ABB RAPID module: P106.mod

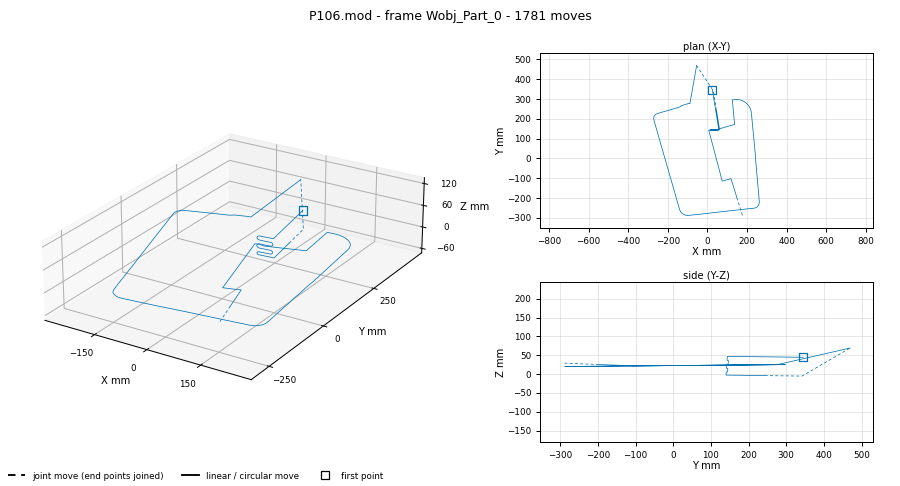
[picture p0: tool path of P106.mod in frame Wobj_Part_0, 1781 of 1791 moves have a stored position in this frame; points joined in program order, loops and branches not executed]
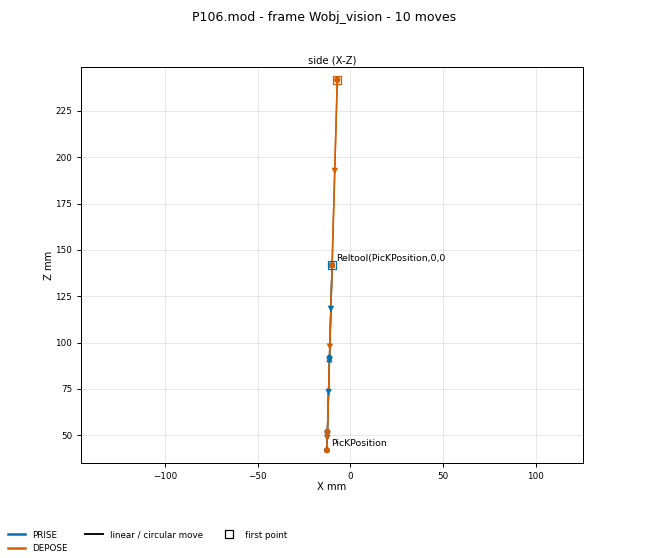
[picture p1: tool path of P106.mod in frame Wobj_vision, 10 of 1791 moves have a stored position in this frame; points joined in program order, loops and branches not executed]
MODULE P106

    ! Nom         :P106
    ! Description :
    ! Créé le     :06/06/2023 16:16:34

    LOCAL CONST SPEEDDATA VitesseLente :=[10,500,0,0];
	LOCAL CONST SPEEDDATA VitesseRapide :=[30,500,0,0];
	LOCAL CONST SPEEDDATA VitesseTronconnage :=[2,500,0,0];
	LOCAL CONST SPEEDDATA VitesseTronconnageApp :=[10,500,0,0];
    !
    !Point de prise
    LOCAL PERS Robtarget PicKPosition := [[-12.6362620334208,-14.9745689455813,41.8593448105357],[-0.00913162142581617,0.993890068091212,0.109216713362201,-0.0130711729443154],[0,0,0,0],[8.999999E+09,8.999999E+09,8.999999E+09,8.999999E+09,8.999999E+09,8.999999E+09]];
	LOCAL PERS Pose Ref := [[0,0,0],[1,0,0,0]];
    !
    !Declaration des points de meulage

    !Tr_meulage_motif_1 : Meulage d'un motif
    LOCAL CONST Robtarget Tr_meulage_motif_1_0 := [[57.250015625,147.518171875,47.0711640625],[0.0569478960959874,-0.0562129652335629,0.700246962774789,-0.709402023393347],[0,0,0,0],[8.999999E+09,8.999999E+09,8.999999E+09,8.999999E+09,8.999999E+09,8.999999E+09]];
    LOCAL CONST Robtarget Tr_meulage_motif_1_1 := [[56.253921875,147.429890625,47.0709765625],[0.0569478960959874,-0.0562129652335629,0.700246962774789,-0.709402023393347],[0,0,0,0],[8.999999E+09,8.999999E+09,8.999999E+09,8.999999E+09,8.999999E+09,8.999999E+09]];
    LOCAL CONST Robtarget Tr_meulage_motif_1_2 := [[55.257828125,147.34159375,47.0707890625],[0.0569478960959874,-0.0562129652335629,0.700246962774789,-0.709402023393347],[0,0,0,0],[8.999999E+09,8.999999E+09,8.999999E+09,8.999999E+09,8.999999E+09,8.999999E+09]];
    LOCAL CONST Robtarget Tr_meulage_motif_1_3 := [[54.261734375,147.253296875,47.07059765625],[0.0569478960959874,-0.0562129652335629,0.700246962774789,-0.709402023393347],[0,0,0,0],[8.999999E+09,8.999999E+09,8.999999E+09,8.999999E+09,8.999999E+09,8.999999E+09]];
    LOCAL CONST Robtarget Tr_meulage_motif_1_4 := [[53.265640625,147.165,47.07041015625],[0.0569478960959874,-0.0562129652335629,0.700246962774789,-0.709402023393347],[0,0,0,0],[8.999999E+09,8.999999E+09,8.999999E+09,8.999999E+09,8.999999E+09,8.999999E+09]];
    LOCAL CONST Robtarget Tr_meulage_motif_1_5 := [[52.269546875,147.076703125,47.07021875],[0.0569478960959874,-0.0562129652335629,0.700246962774789,-0.709402023393347],[0,0,0,0],[8.999999E+09,8.999999E+09,8.999999E+09,8.999999E+09,8.999999E+09,8.999999E+09]];
    LOCAL CONST Robtarget Tr_meulage_motif_1_6 := [[51.27344921875,146.98840625,47.07003125],[0.0569478960959874,-0.0562129652335629,0.700246962774789,-0.709402023393347],[0,0,0,0],[8.999999E+09,8.999999E+09,8.999999E+09,8.999999E+09,8.999999E+09,8.999999E+09]];
    LOCAL CONST Robtarget Tr_meulage_motif_1_7 := [[50.27735546875,146.900125,47.06984375],[0.0569478960959874,-0.0562129652335629,0.700246962774789,-0.709402023393347],[0,0,0,0],[8.999999E+09,8.999999E+09,8.999999E+09,8.999999E+09,8.999999E+09,8.999999E+09]];
    LOCAL CONST Robtarget Tr_meulage_motif_1_8 := [[49.28126171875,146.811828125,47.06965234375],[0.0569478960959874,-0.0562129652335629,0.700246962774789,-0.709402023393347],[0,0,0,0],[8.999999E+09,8.999999E+09,8.999999E+09,8.999999E+09,8.999999E+09,8.999999E+09]];
    LOCAL CONST Robtarget Tr_meulage_motif_1_9 := [[48.28516796875,146.72353125,47.06946484375],[0.0569478960959874,-0.0562129652335629,0.700246962774789,-0.709402023393347],[0,0,0,0],[8.999999E+09,8.999999E+09,8.999999E+09,8.999999E+09,8.999999E+09,8.999999E+09]];
    LOCAL CONST Robtarget Tr_meulage_motif_1_10 := [[47.28907421875,146.635234375,47.0692734375],[0.0569478960959874,-0.0562129652335629,0.700246962774789,-0.709402023393347],[0,0,0,0],[8.999999E+09,8.999999E+09,8.999999E+09,8.999999E+09,8.999999E+09,8.999999E+09]];
    LOCAL CONST Robtarget Tr_meulage_motif_1_11 := [[46.29298046875,146.5469375,47.0690859375],[0.0569478960959874,-0.0562129652335629,0.700246962774789,-0.709402023393347],[0,0,0,0],[8.999999E+09,8.999999E+09,8.999999E+09,8.999999E+09,8.999999E+09,8.999999E+09]];
    LOCAL CONST Robtarget Tr_meulage_motif_1_12 := [[45.2968828125,146.458640625,47.0688984375],[0.0569478960959874,-0.0562129652335629,0.700246962774789,-0.709402023393347],[0,0,0,0],[8.999999E+09,8.999999E+09,8.999999E+09,8.999999E+09,8.999999E+09,8.999999E+09]];
    LOCAL CONST Robtarget Tr_meulage_motif_1_13 := [[44.3007890625,146.370359375,47.06870703125],[0.0569478960959874,-0.0562129652335629,0.700246962774789,-0.709402023393347],[0,0,0,0],[8.999999E+09,8.999999E+09,8.999999E+09,8.999999E+09,8.999999E+09,8.999999E+09]];
    LOCAL CONST Robtarget Tr_meulage_motif_1_14 := [[43.3046953125,146.2820625,47.06851953125],[0.0569478960959874,-0.0562129652335629,0.700246962774789,-0.709402023393347],[0,0,0,0],[8.999999E+09,8.999999E+09,8.999999E+09,8.999999E+09,8.999999E+09,8.999999E+09]];
    LOCAL CONST Robtarget Tr_meulage_motif_1_15 := [[42.3086015625,146.193765625,47.06833203125],[0.0569478960959874,-0.0562129652335629,0.700246962774789,-0.709402023393347],[0,0,0,0],[8.999999E+09,8.999999E+09,8.999999E+09,8.999999E+09,8.999999E+09,8.999999E+09]];
    LOCAL CONST Robtarget Tr_meulage_motif_1_16 := [[41.3125078125,146.10546875,47.068140625],[0.0569478960959874,-0.0562129652335629,0.700246962774789,-0.709402023393347],[0,0,0,0],[8.999999E+09,8.999999E+09,8.999999E+09,8.999999E+09,8.999999E+09,8.999999E+09]];
    LOCAL CONST Robtarget Tr_meulage_motif_1_17 := [[40.31641015625,146.017171875,47.067953125],[0.0569478960959874,-0.0562129652335629,0.700246962774789,-0.709402023393347],[0,0,0,0],[8.999999E+09,8.999999E+09,8.999999E+09,8.999999E+09,8.999999E+09,8.999999E+09]];
    LOCAL CONST Robtarget Tr_meulage_motif_1_18 := [[39.32031640625,145.928875,47.06776171875],[0.0569478960959874,-0.0562129652335629,0.700246962774789,-0.709402023393347],[0,0,0,0],[8.999999E+09,8.999999E+09,8.999999E+09,8.999999E+09,8.999999E+09,8.999999E+09]];
    LOCAL CONST Robtarget Tr_meulage_motif_1_19 := [[38.32422265625,145.84059375,47.06757421875],[0.0569478960959874,-0.0562129652335629,0.700246962774789,-0.709402023393347],[0,0,0,0],[8.999999E+09,8.999999E+09,8.999999E+09,8.999999E+09,8.999999E+09,8.999999E+09]];
    LOCAL CONST Robtarget Tr_meulage_motif_1_20 := [[37.32812890625,145.752296875,47.06738671875],[0.0569478960959874,-0.0562129652335629,0.700246962774789,-0.709402023393347],[0,0,0,0],[8.999999E+09,8.999999E+09,8.999999E+09,8.999999E+09,8.999999E+09,8.999999E+09]];
    LOCAL CONST Robtarget Tr_meulage_motif_1_21 := [[36.33203515625,145.664,47.0671953125],[0.0569478960959874,-0.0562129652335629,0.700246962774789,-0.709402023393347],[0,0,0,0],[8.999999E+09,8.999999E+09,8.999999E+09,8.999999E+09,8.999999E+09,8.999999E+09]];
    LOCAL CONST Robtarget Tr_meulage_motif_1_22 := [[35.33594140625,145.575703125,47.0670078125],[0.0569478960959874,-0.0562129652335629,0.700246962774789,-0.709402023393347],[0,0,0,0],[8.999999E+09,8.999999E+09,8.999999E+09,8.999999E+09,8.999999E+09,8.999999E+09]];
    LOCAL CONST Robtarget Tr_meulage_motif_1_23 := [[34.33984375,145.48740625,47.06681640625],[0.0569478960959874,-0.0562129652335629,0.700246962774789,-0.709402023393347],[0,0,0,0],[8.999999E+09,8.999999E+09,8.999999E+09,8.999999E+09,8.999999E+09,8.999999E+09]];
    LOCAL CONST Robtarget Tr_meulage_motif_1_24 := [[33.34375,145.399125,47.06662890625],[0.0569478960959874,-0.0562129652335629,0.700246962774789,-0.709402023393347],[0,0,0,0],[8.999999E+09,8.999999E+09,8.999999E+09,8.999999E+09,8.999999E+09,8.999999E+09]];
    LOCAL CONST Robtarget Tr_meulage_motif_1_25 := [[32.34765625,145.310828125,47.06644140625],[0.0569478960959874,-0.0562129652335629,0.700246962774789,-0.709402023393347],[0,0,0,0],[8.999999E+09,8.999999E+09,8.999999E+09,8.999999E+09,8.999999E+09,8.999999E+09]];
    LOCAL CONST Robtarget Tr_meulage_motif_1_26 := [[31.3515625,145.22253125,47.06625],[0.0569478960959874,-0.0562129652335629,0.700246962774789,-0.709402023393347],[0,0,0,0],[8.999999E+09,8.999999E+09,8.999999E+09,8.999999E+09,8.999999E+09,8.999999E+09]];
    LOCAL CONST Robtarget Tr_meulage_motif_1_27 := [[30.35546875,145.134234375,47.0660625],[0.0569478960959874,-0.0562129652335629,0.700246962774789,-0.709402023393347],[0,0,0,0],[8.999999E+09,8.999999E+09,8.999999E+09,8.999999E+09,8.999999E+09,8.999999E+09]];
    LOCAL CONST Robtarget Tr_meulage_motif_1_28 := [[29.359373046875,145.0459375,47.06587109375],[0.0569478960959874,-0.0562129652335629,0.700246962774789,-0.709402023393347],[0,0,0,0],[8.999999E+09,8.999999E+09,8.999999E+09,8.999999E+09,8.999999E+09,8.999999E+09]];
    LOCAL CONST Robtarget Tr_meulage_motif_1_29 := [[28.363279296875,144.957640625,47.06568359375],[0.0569478960959874,-0.0562129652335629,0.700246962774789,-0.709402023393347],[0,0,0,0],[8.999999E+09,8.999999E+09,8.999999E+09,8.999999E+09,8.999999E+09,8.999999E+09]];
    LOCAL CONST Robtarget Tr_meulage_motif_1_30 := [[27.36718359375,144.869359375,47.06549609375],[0.0569478960959874,-0.0562129652335629,0.700246962774789,-0.709402023393347],[0,0,0,0],[8.999999E+09,8.999999E+09,8.999999E+09,8.999999E+09,8.999999E+09,8.999999E+09]];
    LOCAL CONST Robtarget Tr_meulage_motif_1_31 := [[26.37108984375,144.7810625,47.0653046875],[0.0569478960959874,-0.0562129652335629,0.700246962774789,-0.709402023393347],[0,0,0,0],[8.999999E+09,8.999999E+09,8.999999E+09,8.999999E+09,8.999999E+09,8.999999E+09]];
    LOCAL CONST Robtarget Tr_meulage_motif_1_32 := [[25.37499609375,144.692765625,47.0651171875],[0.0569478960959874,-0.0562129652335629,0.700246962774789,-0.709402023393347],[0,0,0,0],[8.999999E+09,8.999999E+09,8.999999E+09,8.999999E+09,8.999999E+09,8.999999E+09]];
    LOCAL CONST Robtarget Tr_meulage_motif_1_33 := [[24.378900390625,144.60446875,47.06492578125],[0.0569478960959874,-0.0562129652335629,0.700246962774789,-0.709402023393347],[0,0,0,0],[8.999999E+09,8.999999E+09,8.999999E+09,8.999999E+09,8.999999E+09,8.999999E+09]];
    LOCAL CONST Robtarget Tr_meulage_motif_1_34 := [[23.382806640625,144.516171875,47.06473828125],[0.0569478960959874,-0.0562129652335629,0.700246962774789,-0.709402023393347],[0,0,0,0],[8.999999E+09,8.999999E+09,8.999999E+09,8.999999E+09,8.999999E+09,8.999999E+09]];
    LOCAL CONST Robtarget Tr_meulage_motif_1_35 := [[22.386712890625,144.427875,47.06455078125],[0.0569478960959874,-0.0562129652335629,0.700246962774789,-0.709402023393347],[0,0,0,0],[8.999999E+09,8.999999E+09,8.999999E+09,8.999999E+09,8.999999E+09,8.999999E+09]];
    LOCAL CONST Robtarget Tr_meulage_motif_1_36 := [[21.3906171875,144.33959375,47.064359375],[0.0569478960959874,-0.0562129652335629,0.700246962774789,-0.709402023393347],[0,0,0,0],[8.999999E+09,8.999999E+09,8.999999E+09,8.999999E+09,8.999999E+09,8.999999E+09]];
    LOCAL CONST Robtarget Tr_meulage_motif_1_37 := [[20.3945234375,144.251296875,47.064171875],[0.0569478960959874,-0.0562129652335629,0.700246962774789,-0.709402023393347],[0,0,0,0],[8.999999E+09,8.999999E+09,8.999999E+09,8.999999E+09,8.999999E+09,8.999999E+09]];
    LOCAL CONST Robtarget Tr_meulage_motif_1_38 := [[19.3984296875,144.163,47.06398046875],[0.0569478960959874,-0.0562129652335629,0.700246962774789,-0.709402023393347],[0,0,0,0],[8.999999E+09,8.999999E+09,8.999999E+09,8.999999E+09,8.999999E+09,8.999999E+09]];
    LOCAL CONST Robtarget Tr_meulage_motif_1_39 := [[18.41045703125,144.067546875,46.95348046875],[0.0569478960959874,-0.0562129652335629,0.700246962774789,-0.709402023393347],[0,0,0,0],[8.999999E+09,8.999999E+09,8.999999E+09,8.999999E+09,8.999999E+09,8.999999E+09]];
    LOCAL CONST Robtarget Tr_meulage_motif_1_40 := [[17.469013671875,143.969078125,46.74264453125],[0.0569478960959874,-0.0562129652335629,0.700246962774789,-0.709402023393347],[0,0,0,0],[8.999999E+09,8.999999E+09,8.999999E+09,8.999999E+09,8.999999E+09,8.999999E+09]];
    LOCAL CONST Robtarget Tr_meulage_motif_1_41 := [[16.62137890625,143.87459375,46.47132421875],[0.0569478960959874,-0.0562129652335629,0.700246962774789,-0.709402023393347],[0,0,0,0],[8.999999E+09,8.999999E+09,8.999999E+09,8.999999E+09,8.999999E+09,8.999999E+09]];
    LOCAL CONST Robtarget Tr_meulage_motif_1_42 := [[15.8761484375,143.78890625,46.1959375],[0.0569478960959874,-0.0562129652335629,0.700246962774789,-0.709402023393347],[0,0,0,0],[8.999999E+09,8.999999E+09,8.999999E+09,8.999999E+09,8.999999E+09,8.999999E+09]];
    LOCAL CONST Robtarget Tr_meulage_motif_1_43 := [[14.7833583984375,143.6481875,45.58115234375],[0.0569478960959874,-0.0562129652335629,0.700246962774789,-0.709402023393347],[0,0,0,0],[8.999999E+09,8.999999E+09,8.999999E+09,8.999999E+09,8.999999E+09,8.999999E+09]];
    LOCAL CONST Robtarget Tr_meulage_motif_1_44 := [[13.768947265625,143.497953125,44.7354375],[0.0569478960959874,-0.0562129652335629,0.700246962774789,-0.709402023393347],[0,0,0,0],[8.999999E+09,8.999999E+09,8.999999E+09,8.999999E+09,8.999999E+09,8.999999E+09]];
    LOCAL CONST Robtarget Tr_meulage_motif_1_45 := [[12.9312021484375,143.350828125,43.7139765625],[0.0569478960959874,-0.0562129652335629,0.700246962774789,-0.709402023393347],[0,0,0,0],[8.999999E+09,8.999999E+09,8.999999E+09,8.999999E+09,8.999999E+09,8.999999E+09]];
    LOCAL CONST Robtarget Tr_meulage_motif_1_46 := [[12.4521484375,143.228921875,42.60050390625],[0.0569478960959874,-0.0562129652335629,0.700246962774789,-0.709402023393347],[0,0,0,0],[8.999999E+09,8.999999E+09,8.999999E+09,8.999999E+09,8.999999E+09,8.999999E+09]];
    LOCAL CONST Robtarget Tr_meulage_motif_1_47 := [[12.429677734375,143.17740625,41.90628125],[0.0569478960959874,-0.0562129652335629,0.700246962774789,-0.709402023393347],[0,0,0,0],[8.999999E+09,8.999999E+09,8.999999E+09,8.999999E+09,8.999999E+09,8.999999E+09]];
    LOCAL CONST Robtarget Tr_meulage_motif_1_48 := [[12.43394140625,143.13071875,41.2466953125],[0.0569478960959874,-0.0562129652335629,0.700246962774789,-0.709402023393347],[0,0,0,0],[8.999999E+09,8.999999E+09,8.999999E+09,8.999999E+09,8.999999E+09,8.999999E+09]];
    LOCAL CONST Robtarget Tr_meulage_motif_1_49 := [[12.49286328125,143.08890625,40.58727734375],[0.0569478960959874,-0.0562129652335629,0.700246962774789,-0.709402023393347],[0,0,0,0],[8.999999E+09,8.999999E+09,8.999999E+09,8.999999E+09,8.999999E+09,8.999999E+09]];
    LOCAL CONST Robtarget Tr_meulage_motif_1_50 := [[12.9962392578125,143.055109375,39.488390625],[0.0569478960959874,-0.0562129652335629,0.700246962774789,-0.709402023393347],[0,0,0,0],[8.999999E+09,8.999999E+09,8.999999E+09,8.999999E+09,8.999999E+09,8.999999E+09]];
    LOCAL CONST Robtarget Tr_meulage_motif_1_51 := [[13.8560078125,143.0596875,38.4844609375],[0.0569478960959874,-0.0562129652335629,0.700246962774789,-0.709402023393347],[0,0,0,0],[8.999999E+09,8.999999E+09,8.999999E+09,8.999999E+09,8.999999E+09,8.999999E+09]];
    LOCAL CONST Robtarget Tr_meulage_motif_1_52 := [[14.8807607421875,143.09153125,37.65786328125],[0.0569478960959874,-0.0562129652335629,0.700246962774789,-0.709402023393347],[0,0,0,0],[8.999999E+09,8.999999E+09,8.999999E+09,8.999999E+09,8.999999E+09,8.999999E+09]];
    LOCAL CONST Robtarget Tr_meulage_motif_1_53 := [[15.56772265625,143.124265625,37.26323828125],[0.0569478960959874,-0.0562129652335629,0.700246962774789,-0.709402023393347],[0,0,0,0],[8.999999E+09,8.999999E+09,8.999999E+09,8.999999E+09,8.999999E+09,8.999999E+09]];
    LOCAL CONST Robtarget Tr_meulage_motif_1_54 := [[16.724498046875,143.192109375,36.77715234375],[0.0569478960959874,-0.0562129652335629,0.700246962774789,-0.709402023393347],[0,0,0,0],[8.999999E+09,8.999999E+09,8.999999E+09,8.999999E+09,8.999999E+09,8.999999E+09]];
    LOCAL CONST Robtarget Tr_meulage_motif_1_55 := [[17.567931640625,143.248078125,36.5138828125],[0.0569478960959874,-0.0562129652335629,0.700246962774789,-0.709402023393347],[0,0,0,0],[8.999999E+09,8.999999E+09,8.999999E+09,8.999999E+09,8.999999E+09,8.999999E+09]];
    LOCAL CONST Robtarget Tr_meulage_motif_1_56 := [[18.497609375,143.3159375,36.31010546875],[0.0569478960959874,-0.0562129652335629,0.700246962774789,-0.709402023393347],[0,0,0,0],[8.999999E+09,8.999999E+09,8.999999E+09,8.999999E+09,8.999999E+09,8.999999E+09]];
    LOCAL CONST Robtarget Tr_meulage_motif_1_57 := [[19.4760390625,143.3949375,36.20197265625],[0.0569478960959874,-0.0562129652335629,0.700246962774789,-0.709402023393347],[0,0,0,0],[8.999999E+09,8.999999E+09,8.999999E+09,8.999999E+09,8.999999E+09,8.999999E+09]];
    LOCAL CONST Robtarget Tr_meulage_motif_1_58 := [[20.4654375,143.474765625,36.09184375],[0.0569478960959874,-0.0562129652335629,0.700246962774789,-0.709402023393347],[0,0,0,0],[8.999999E+09,8.999999E+09,8.999999E+09,8.999999E+09,8.999999E+09,8.999999E+09]];
    LOCAL CONST Robtarget Tr_meulage_motif_1_59 := [[21.461533203125,143.5630625,36.09203125],[0.0569478960959874,-0.0562129652335629,0.700246962774789,-0.709402023393347],[0,0,0,0],[8.999999E+09,8.999999E+09,8.999999E+09,8.999999E+09,8.999999E+09,8.999999E+09]];
    LOCAL CONST Robtarget Tr_meulage_motif_1_60 := [[22.457626953125,143.65134375,36.09222265625],[0.0569478960959874,-0.0562129652335629,0.700246962774789,-0.709402023393347],[0,0,0,0],[8.999999E+09,8.999999E+09,8.999999E+09,8.999999E+09,8.999999E+09,8.999999E+09]];
    LOCAL CONST Robtarget Tr_meulage_motif_1_61 := [[23.453720703125,143.739640625,36.09241015625],[0.0569478960959874,-0.0562129652335629,0.700246962774789,-0.709402023393347],[0,0,0,0],[8.999999E+09,8.999999E+09,8.999999E+09,8.999999E+09,8.999999E+09,8.999999E+09]];
    LOCAL CONST Robtarget Tr_meulage_motif_1_62 := [[24.44981640625,143.8279375,36.0926015625],[0.0569478960959874,-0.0562129652335629,0.700246962774789,-0.709402023393347],[0,0,0,0],[8.999999E+09,8.999999E+09,8.999999E+09,8.999999E+09,8.999999E+09,8.999999E+09]];
    LOCAL CONST Robtarget Tr_meulage_motif_1_63 := [[25.44591015625,143.916234375,36.0927890625],[0.0569478960959874,-0.0562129652335629,0.700246962774789,-0.709402023393347],[0,0,0,0],[8.999999E+09,8.999999E+09,8.999999E+09,8.999999E+09,8.999999E+09,8.999999E+09]];
    LOCAL CONST Robtarget Tr_meulage_motif_1_64 := [[26.44200390625,144.00453125,36.0929765625],[0.0569478960959874,-0.0562129652335629,0.700246962774789,-0.709402023393347],[0,0,0,0],[8.999999E+09,8.999999E+09,8.999999E+09,8.999999E+09,8.999999E+09,8.999999E+09]];
    LOCAL CONST Robtarget Tr_meulage_motif_1_65 := [[27.438099609375,144.092828125,36.09316796875],[0.0569478960959874,-0.0562129652335629,0.700246962774789,-0.709402023393347],[0,0,0,0],[8.999999E+09,8.999999E+09,8.999999E+09,8.999999E+09,8.999999E+09,8.999999E+09]];
    LOCAL CONST Robtarget Tr_meulage_motif_1_66 := [[28.434193359375,144.181109375,36.09335546875],[0.0569478960959874,-0.0562129652335629,0.700246962774789,-0.709402023393347],[0,0,0,0],[8.999999E+09,8.999999E+09,8.999999E+09,8.999999E+09,8.999999E+09,8.999999E+09]];
    LOCAL CONST Robtarget Tr_meulage_motif_1_67 := [[29.430287109375,144.26940625,36.093546875],[0.0569478960959874,-0.0562129652335629,0.700246962774789,-0.709402023393347],[0,0,0,0],[8.999999E+09,8.999999E+09,8.999999E+09,8.999999E+09,8.999999E+09,8.999999E+09]];
    LOCAL CONST Robtarget Tr_meulage_motif_1_68 := [[30.4263828125,144.357703125,36.093734375],[0.0569478960959874,-0.0562129652335629,0.700246962774789,-0.709402023393347],[0,0,0,0],[8.999999E+09,8.999999E+09,8.999999E+09,8.999999E+09,8.999999E+09,8.999999E+09]];
    LOCAL CONST Robtarget Tr_meulage_motif_1_69 := [[31.4224765625,144.446,36.093921875],[0.0569478960959874,-0.0562129652335629,0.700246962774789,-0.709402023393347],[0,0,0,0],[8.999999E+09,8.999999E+09,8.999999E+09,8.999999E+09,8.999999E+09,8.999999E+09]];
    LOCAL CONST Robtarget Tr_meulage_motif_1_70 := [[32.4185703125,144.534296875,36.09411328125],[0.0569478960959874,-0.0562129652335629,0.700246962774789,-0.709402023393347],[0,0,0,0],[8.999999E+09,8.999999E+09,8.999999E+09,8.999999E+09,8.999999E+09,8.999999E+09]];
    LOCAL CONST Robtarget Tr_meulage_motif_1_71 := [[33.4146640625,144.622578125,36.09430078125],[0.0569478960959874,-0.0562129652335629,0.700246962774789,-0.709402023393347],[0,0,0,0],[8.999999E+09,8.999999E+09,8.999999E+09,8.999999E+09,8.999999E+09,8.999999E+09]];
    LOCAL CONST Robtarget Tr_meulage_motif_1_72 := [[34.41076171875,144.710875,36.09448828125],[0.0569478960959874,-0.0562129652335629,0.700246962774789,-0.709402023393347],[0,0,0,0],[8.999999E+09,8.999999E+09,8.999999E+09,8.999999E+09,8.999999E+09,8.999999E+09]];
    LOCAL CONST Robtarget Tr_meulage_motif_1_73 := [[35.40685546875,144.799171875,36.0946796875],[0.0569478960959874,-0.0562129652335629,0.700246962774789,-0.709402023393347],[0,0,0,0],[8.999999E+09,8.999999E+09,8.999999E+09,8.999999E+09,8.999999E+09,8.999999E+09]];
    LOCAL CONST Robtarget Tr_meulage_motif_1_74 := [[36.40294921875,144.88746875,36.0948671875],[0.0569478960959874,-0.0562129652335629,0.700246962774789,-0.709402023393347],[0,0,0,0],[8.999999E+09,8.999999E+09,8.999999E+09,8.999999E+09,8.999999E+09,8.999999E+09]];
    LOCAL CONST Robtarget Tr_meulage_motif_1_75 := [[37.39904296875,144.975765625,36.09505859375],[0.0569478960959874,-0.0562129652335629,0.700246962774789,-0.709402023393347],[0,0,0,0],[8.999999E+09,8.999999E+09,8.999999E+09,8.999999E+09,8.999999E+09,8.999999E+09]];
    LOCAL CONST Robtarget Tr_meulage_motif_1_76 := [[38.39513671875,145.0640625,36.09524609375],[0.0569478960959874,-0.0562129652335629,0.700246962774789,-0.709402023393347],[0,0,0,0],[8.999999E+09,8.999999E+09,8.999999E+09,8.999999E+09,8.999999E+09,8.999999E+09]];
    LOCAL CONST Robtarget Tr_meulage_motif_1_77 := [[39.39123046875,145.15234375,36.09543359375],[0.0569478960959874,-0.0562129652335629,0.700246962774789,-0.709402023393347],[0,0,0,0],[8.999999E+09,8.999999E+09,8.999999E+09,8.999999E+09,8.999999E+09,8.999999E+09]];
    LOCAL CONST Robtarget Tr_meulage_motif_1_78 := [[40.387328125,145.240640625,36.095625],[0.0569478960959874,-0.0562129652335629,0.700246962774789,-0.709402023393347],[0,0,0,0],[8.999999E+09,8.999999E+09,8.999999E+09,8.999999E+09,8.999999E+09,8.999999E+09]];
    LOCAL CONST Robtarget Tr_meulage_motif_1_79 := [[41.383421875,145.3289375,36.0958125],[0.0569478960959874,-0.0562129652335629,0.700246962774789,-0.709402023393347],[0,0,0,0],[8.999999E+09,8.999999E+09,8.999999E+09,8.999999E+09,8.999999E+09,8.999999E+09]];
    LOCAL CONST Robtarget Tr_meulage_motif_1_80 := [[42.379515625,145.417234375,36.09600390625],[0.0569478960959874,-0.0562129652335629,0.700246962774789,-0.709402023393347],[0,0,0,0],[8.999999E+09,8.999999E+09,8.999999E+09,8.999999E+09,8.999999E+09,8.999999E+09]];
    LOCAL CONST Robtarget Tr_meulage_motif_1_81 := [[43.375609375,145.50553125,36.09619140625],[0.0569478960959874,-0.0562129652335629,0.700246962774789,-0.709402023393347],[0,0,0,0],[8.999999E+09,8.999999E+09,8.999999E+09,8.999999E+09,8.999999E+09,8.999999E+09]];
    LOCAL CONST Robtarget Tr_meulage_motif_1_82 := [[44.371703125,145.593828125,36.09637890625],[0.0569478960959874,-0.0562129652335629,0.700246962774789,-0.709402023393347],[0,0,0,0],[8.999999E+09,8.999999E+09,8.999999E+09,8.999999E+09,8.999999E+09,8.999999E+09]];
    LOCAL CONST Robtarget Tr_meulage_motif_1_83 := [[45.367796875,145.682109375,36.0965703125],[0.0569478960959874,-0.0562129652335629,0.700246962774789,-0.709402023393347],[0,0,0,0],[8.999999E+09,8.999999E+09,8.999999E+09,8.999999E+09,8.999999E+09,8.999999E+09]];
    LOCAL CONST Robtarget Tr_meulage_motif_1_84 := [[46.36389453125,145.77040625,36.0967578125],[0.0569478960959874,-0.0562129652335629,0.700246962774789,-0.709402023393347],[0,0,0,0],[8.999999E+09,8.999999E+09,8.999999E+09,8.999999E+09,8.999999E+09,8.999999E+09]];
    LOCAL CONST Robtarget Tr_meulage_motif_1_85 := [[47.35998828125,145.858703125,36.09694921875],[0.0569478960959874,-0.0562129652335629,0.700246962774789,-0.709402023393347],[0,0,0,0],[8.999999E+09,8.999999E+09,8.999999E+09,8.999999E+09,8.999999E+09,8.999999E+09]];
    LOCAL CONST Robtarget Tr_meulage_motif_1_86 := [[48.35608203125,145.947,36.09713671875],[0.0569478960959874,-0.0562129652335629,0.700246962774789,-0.709402023393347],[0,0,0,0],[8.999999E+09,8.999999E+09,8.999999E+09,8.999999E+09,8.999999E+09,8.999999E+09]];
    LOCAL CONST Robtarget Tr_meulage_motif_1_87 := [[49.35217578125,146.035296875,36.09732421875],[0.0569478960959874,-0.0562129652335629,0.700246962774789,-0.709402023393347],[0,0,0,0],[8.999999E+09,8.999999E+09,8.999999E+09,8.999999E+09,8.999999E+09,8.999999E+09]];
    LOCAL CONST Robtarget Tr_meulage_motif_1_88 := [[50.34826953125,146.12359375,36.097515625],[0.0569478960959874,-0.0562129652335629,0.700246962774789,-0.709402023393347],[0,0,0,0],[8.999999E+09,8.999999E+09,8.999999E+09,8.999999E+09,8.999999E+09,8.999999E+09]];
    LOCAL CONST Robtarget Tr_meulage_motif_1_89 := [[51.33766796875,146.203421875,35.98738671875],[0.0569478960959874,-0.0562129652335629,0.700246962774789,-0.709402023393347],[0,0,0,0],[8.999999E+09,8.999999E+09,8.999999E+09,8.999999E+09,8.999999E+09,8.999999E+09]];
    LOCAL CONST Robtarget Tr_meulage_motif_1_90 := [[52.2818359375,146.272078125,35.77691015625],[0.0569478960959874,-0.0562129652335629,0.700246962774789,-0.709402023393347],[0,0,0,0],[8.999999E+09,8.999999E+09,8.999999E+09,8.999999E+09,8.999999E+09,8.999999E+09]];
    LOCAL CONST Robtarget Tr_meulage_motif_1_91 := [[53.1329765625,146.328171875,35.50591015625],[0.0569478960959874,-0.0562129652335629,0.700246962774789,-0.709402023393347],[0,0,0,0],[8.999999E+09,8.999999E+09,8.999999E+09,8.999999E+09,8.999999E+09,8.999999E+09]];
    LOCAL CONST Robtarget Tr_meulage_motif_1_92 := [[53.84365625,146.36953125,35.20265625],[0.0569478960959874,-0.0562129652335629,0.700246962774789,-0.709402023393347],[0,0,0,0],[8.999999E+09,8.999999E+09,8.999999E+09,8.999999E+09,8.999999E+09,8.999999E+09]];
    LOCAL CONST Robtarget Tr_meulage_motif_1_93 := [[54.87835546875,146.41409375,34.541984375],[0.0569478960959874,-0.0562129652335629,0.700246962774789,-0.709402023393347],[0,0,0,0],[8.999999E+09,8.999999E+09,8.999999E+09,8.999999E+09,8.999999E+09,8.999999E+09]];
    LOCAL CONST Robtarget Tr_meulage_motif_1_94 := [[55.7825859375,146.4300625,33.64248828125],[0.0569478960959874,-0.0562129652335629,0.700246962774789,-0.709402023393347],[0,0,0,0],[8.999999E+09,8.999999E+09,8.999999E+09,8.999999E+09,8.999999E+09,8.999999E+09]];
    LOCAL CONST Robtarget Tr_meulage_motif_1_95 := [[56.3222109375,146.403453125,32.599189453125],[0.0569478960959874,-0.0562129652335629,0.700246962774789,-0.709402023393347],[0,0,0,0],[8.999999E+09,8.999999E+09,8.999999E+09,8.999999E+09,8.999999E+09,8.999999E+09]];
    LOCAL CONST Robtarget Tr_meulage_motif_1_96 := [[56.51073828125,146.370828125,31.90775],[0.0569478960959874,-0.0562129652335629,0.700246962774789,-0.709402023393347],[0,0,0,0],[8.999999E+09,8.999999E+09,8.999999E+09,8.999999E+09,8.999999E+09,8.999999E+09]];
    LOCAL CONST Robtarget Tr_meulage_motif_1_97 := [[56.579296875,146.322109375,31.13969921875],[0.0569478960959874,-0.0562129652335629,0.700246962774789,-0.709402023393347],[0,0,0,0],[8.999999E+09,8.999999E+09,8.999999E+09,8.999999E+09,8.999999E+09,8.999999E+09]];
    LOCAL CONST Robtarget Tr_meulage_motif_1_98 := [[56.51758203125,146.26184375,30.371748046875],[0.0569478960959874,-0.0562129652335629,0.700246962774789,-0.709402023393347],[0,0,0,0],[8.999999E+09,8.999999E+09,8.999999E+09,8.999999E+09,8.999999E+09,8.999999E+09]];
    LOCAL CONST Robtarget Tr_meulage_motif_1_99 := [[56.1067734375,146.1465625,29.26620703125],[0.0569478960959874,-0.0562129652335629,0.700246962774789,-0.709402023393347],[0,0,0,0],[8.999999E+09,8.999999E+09,8.999999E+09,8.999999E+09,8.999999E+09,8.999999E+09]];
    LOCAL CONST Robtarget Tr_meulage_motif_1_100 := [[55.69785546875,146.068640625,28.6819140625],[0.0569478960959874,-0.0562129652335629,0.700246962774789,-0.709402023393347],[0,0,0,0],[8.999999E+09,8.999999E+09,8.999999E+09,8.999999E+09,8.999999E+09,8.999999E+09]];
    LOCAL CONST Robtarget Tr_meulage_motif_1_101 := [[54.8199140625,145.9276875,27.796853515625],[0.0569478960959874,-0.0562129652335629,0.700246962774789,-0.709402023393347],[0,0,0,0],[8.999999E+09,8.999999E+09,8.999999E+09,8.999999E+09,8.999999E+09,8.999999E+09]];
    LOCAL CONST Robtarget Tr_meulage_motif_1_102 := [[54.23918359375,145.84671875,27.38347265625],[0.0569478960959874,-0.0562129652335629,0.700246962774789,-0.709402023393347],[0,0,0,0],[8.999999E+09,8.999999E+09,8.999999E+09,8.999999E+09,8.999999E+09,8.999999E+09]];
    LOCAL CONST Robtarget Tr_meulage_motif_1_103 := [[53.12915234375,145.709609375,26.84053515625],[0.0569478960959874,-0.0562129652335629,0.700246962774789,-0.709402023393347],[0,0,0,0],[8.999999E+09,8.999999E+09,8.999999E+09,8.999999E+09,8.999999E+09,8.999999E+09]];
    LOCAL CONST Robtarget Tr_meulage_motif_1_104 := [[52.3086875,145.615859375,26.545623046875],[0.0569478960959874,-0.0562129652335629,0.700246962774789,-0.709402023393347],[0,0,0,0],[8.999999E+09,8.999999E+09,8.999999E+09,8.999999E+09,8.999999E+09,8.999999E+09]];
    LOCAL CONST Robtarget Tr_meulage_motif_1_105 := [[51.38164453125,145.519125,26.3414921875],[0.0569478960959874,-0.0562129652335629,0.700246962774789,-0.709402023393347],[0,0,0,0],[8.999999E+09,8.999999E+09,8.999999E+09,8.999999E+09,8.999999E+09,8.999999E+09]];
    LOCAL CONST Robtarget Tr_meulage_motif_1_106 := [[50.4046171875,145.424796875,26.232986328125],[0.0569478960959874,-0.0562129652335629,0.700246962774789,-0.709402023393347],[0,0,0,0],[8.999999E+09,8.999999E+09,8.999999E+09,8.999999E+09,8.999999E+09,8.999999E+09]];
    LOCAL CONST Robtarget Tr_meulage_motif_1_107 := [[49.41664453125,145.329359375,26.122482421875],[0.0569478960959874,-0.0562129652335629,0.700246962774789,-0.709402023393347],[0,0,0,0],[8.999999E+09,8.999999E+09,8.999999E+09,8.999999E+09,8.999999E+09,8.999999E+09]];
    LOCAL CONST Robtarget Tr_meulage_motif_1_108 := [[48.42055078125,145.2410625,26.12229296875],[0.0569478960959874,-0.0562129652335629,0.700246962774789,-0.709402023393347],[0,0,0,0],[8.999999E+09,8.999999E+09,8.999999E+09,8.999999E+09,8.999999E+09,8.999999E+09]];
    LOCAL CONST Robtarget Tr_meulage_motif_1_109 := [[47.42445703125,145.152765625,26.12210546875],[0.0569478960959874,-0.0562129652335629,0.700246962774789,-0.709402023393347],[0,0,0,0],[8.999999E+09,8.999999E+09,8.999999E+09,8.999999E+09,8.999999E+09,8.999999E+09]];
    LOCAL CONST Robtarget Tr_meulage_motif_1_110 := [[46.428359375,145.06446875,26.121916015625],[0.0569478960959874,-0.0562129652335629,0.700246962774789,-0.709402023393347],[0,0,0,0],[8.999999E+09,8.999999E+09,8.999999E+09,8.999999E+09,8.999999E+09,8.999999E+09]];
    LOCAL CONST Robtarget Tr_meulage_motif_1_111 := [[45.432265625,144.976171875,26.1217265625],[0.0569478960959874,-0.0562129652335629,0.700246962774789,-0.709402023393347],[0,0,0,0],[8.999999E+09,8.999999E+09,8.999999E+09,8.999999E+09,8.999999E+09,8.999999E+09]];
    LOCAL CONST Robtarget Tr_meulage_motif_1_112 := [[44.436171875,144.887890625,26.121537109375],[0.0569478960959874,-0.0562129652335629,0.700246962774789,-0.709402023393347],[0,0,0,0],[8.999999E+09,8.999999E+09,8.999999E+09,8.999999E+09,8.999999E+09,8.999999E+09]];
    LOCAL CONST Robtarget Tr_meulage_motif_1_113 := [[43.440078125,144.79959375,26.12134765625],[0.0569478960959874,-0.0562129652335629,0.700246962774789,-0.709402023393347],[0,0,0,0],[8.999999E+09,8.999999E+09,8.999999E+09,8.999999E+09,8.999999E+09,8.999999E+09]];
    LOCAL CONST Robtarget Tr_meulage_motif_1_114 := [[42.443984375,144.711296875,26.12116015625],[0.0569478960959874,-0.0562129652335629,0.700246962774789,-0.709402023393347],[0,0,0,0],[8.999999E+09,8.999999E+09,8.999999E+09,8.999999E+09,8.999999E+09,8.999999E+09]];
    LOCAL CONST Robtarget Tr_meulage_motif_1_115 := [[41.447890625,144.623,26.120970703125],[0.0569478960959874,-0.0562129652335629,0.700246962774789,-0.709402023393347],[0,0,0,0],[8.999999E+09,8.999999E+09,8.999999E+09,8.999999E+09,8.999999E+09,8.999999E+09]];
    LOCAL CONST Robtarget Tr_meulage_motif_1_116 := [[40.45179296875,144.534703125,26.12078125],[0.0569478960959874,-0.0562129652335629,0.700246962774789,-0.709402023393347],[0,0,0,0],[8.999999E+09,8.999999E+09,8.999999E+09,8.999999E+09,8.999999E+09,8.999999E+09]];
    LOCAL CONST Robtarget Tr_meulage_motif_1_117 := [[39.45569921875,144.44640625,26.120591796875],[0.0569478960959874,-0.0562129652335629,0.700246962774789,-0.709402023393347],[0,0,0,0],[8.999999E+09,8.999999E+09,8.999999E+09,8.999999E+09,8.999999E+09,8.999999E+09]];
    LOCAL CONST Robtarget Tr_meulage_motif_1_118 := [[38.45960546875,144.358125,26.12040234375],[0.0569478960959874,-0.0562129652335629,0.700246962774789,-0.709402023393347],[0,0,0,0],[8.999999E+09,8.999999E+09,8.999999E+09,8.999999E+09,8.999999E+09,8.999999E+09]];
    LOCAL CONST Robtarget Tr_meulage_motif_1_119 := [[37.46351171875,144.269828125,26.12021484375],[0.0569478960959874,-0.0562129652335629,0.700246962774789,-0.709402023393347],[0,0,0,0],[8.999999E+09,8.999999E+09,8.999999E+09,8.999999E+09,8.999999E+09,8.999999E+09]];
    LOCAL CONST Robtarget Tr_meulage_motif_1_120 := [[36.46741796875,144.18153125,26.120025390625],[0.0569478960959874,-0.0562129652335629,0.700246962774789,-0.709402023393347],[0,0,0,0],[8.999999E+09,8.999999E+09,8.999999E+09,8.999999E+09,8.999999E+09,8.999999E+09]];
    LOCAL CONST Robtarget Tr_meulage_motif_1_121 := [[35.4713203125,144.093234375,26.1198359375],[0.0569478960959874,-0.0562129652335629,0.700246962774789,-0.709402023393347],[0,0,0,0],[8.999999E+09,8.999999E+09,8.999999E+09,8.999999E+09,8.999999E+09,8.999999E+09]];
    LOCAL CONST Robtarget Tr_meulage_motif_1_122 := [[34.4752265625,144.0049375,26.119646484375],[0.0569478960959874,-0.0562129652335629,0.700246962774789,-0.709402023393347],[0,0,0,0],[8.999999E+09,8.999999E+09,8.999999E+09,8.999999E+09,8.999999E+09,8.999999E+09]];
    LOCAL CONST Robtarget Tr_meulage_motif_1_123 := [[33.4791328125,143.916640625,26.119458984375],[0.0569478960959874,-0.0562129652335629,0.700246962774789,-0.709402023393347],[0,0,0,0],[8.999999E+09,8.999999E+09,8.999999E+09,8.999999E+09,8.999999E+09,8.999999E+09]];
    LOCAL CONST Robtarget Tr_meulage_motif_1_124 := [[32.4830390625,143.828359375,26.11926953125],[0.0569478960959874,-0.0562129652335629,0.700246962774789,-0.709402023393347],[0,0,0,0],[8.999999E+09,8.999999E+09,8.999999E+09,8.999999E+09,8.999999E+09,8.999999E+09]];
    LOCAL CONST Robtarget Tr_meulage_motif_1_125 := [[31.4869453125,143.7400625,26.119080078125],[0.0569478960959874,-0.0562129652335629,0.700246962774789,-0.709402023393347],[0,0,0,0],[8.999999E+09,8.999999E+09,8.999999E+09,8.999999E+09,8.999999E+09,8.999999E+09]];
    LOCAL CONST Robtarget Tr_meulage_motif_1_126 := [[30.490849609375,143.651765625,26.118890625],[0.0569478960959874,-0.0562129652335629,0.700246962774789,-0.709402023393347],[0,0,0,0],[8.999999E+09,8.999999E+09,8.999999E+09,8.999999E+09,8.999999E+09,8.999999E+09]];
    LOCAL CONST Robtarget Tr_meulage_motif_1_127 := [[29.494755859375,143.56346875,26.118701171875],[0.0569478960959874,-0.0562129652335629,0.700246962774789,-0.709402023393347],[0,0,0,0],[8.999999E+09,8.999999E+09,8.999999E+09,8.999999E+09,8.999999E+09,8.999999E+09]];
    LOCAL CONST Robtarget Tr_meulage_motif_1_128 := [[28.498662109375,143.475171875,26.118513671875],[0.0569478960959874,-0.0562129652335629,0.700246962774789,-0.709402023393347],[0,0,0,0],[8.999999E+09,8.999999E+09,8.999999E+09,8.999999E+09,8.999999E+09,8.999999E+09]];
    LOCAL CONST Robtarget Tr_meulage_motif_1_129 := [[27.50256640625,143.386875,26.11832421875],[0.0569478960959874,-0.0562129652335629,0.700246962774789,-0.709402023393347],[0,0,0,0],[8.999999E+09,8.999999E+09,8.999999E+09,8.999999E+09,8.999999E+09,8.999999E+09]];
    LOCAL CONST Robtarget Tr_meulage_motif_1_130 := [[26.50647265625,143.29859375,26.118134765625],[0.0569478960959874,-0.0562129652335629,0.700246962774789,-0.709402023393347],[0,0,0,0],[8.999999E+09,8.999999E+09,8.999999E+09,8.999999E+09,8.999999E+09,8.999999E+09]];
    LOCAL CONST Robtarget Tr_meulage_motif_1_131 := [[25.51037890625,143.210296875,26.1179453125],[0.0569478960959874,-0.0562129652335629,0.700246962774789,-0.709402023393347],[0,0,0,0],[8.999999E+09,8.999999E+09,8.999999E+09,8.999999E+09,8.999999E+09,8.999999E+09]];
    LOCAL CONST Robtarget Tr_meulage_motif_1_132 := [[24.514283203125,143.122,26.117755859375],[0.0569478960959874,-0.0562129652335629,0.700246962774789,-0.709402023393347],[0,0,0,0],[8.999999E+09,8.999999E+09,8.999999E+09,8.999999E+09,8.999999E+09,8.999999E+09]];
    LOCAL CONST Robtarget Tr_meulage_motif_1_133 := [[23.518189453125,143.033703125,26.117568359375],[0.0569478960959874,-0.0562129652335629,0.700246962774789,-0.709402023393347],[0,0,0,0],[8.999999E+09,8.999999E+09,8.999999E+09,8.999999E+09,8.999999E+09,8.999999E+09]];
    LOCAL CONST Robtarget Tr_meulage_motif_1_134 := [[22.522095703125,142.94540625,26.11737890625],[0.0569478960959874,-0.0562129652335629,0.700246962774789,-0.709402023393347],[0,0,0,0],[8.999999E+09,8.999999E+09,8.999999E+09,8.999999E+09,8.999999E+09,8.999999E+09]];
    LOCAL CONST Robtarget Tr_meulage_motif_1_135 := [[21.526,142.857125,26.117189453125],[0.0569478960959874,-0.0562129652335629,0.700246962774789,-0.709402023393347],[0,0,0,0],[8.999999E+09,8.999999E+09,8.999999E+09,8.999999E+09,8.999999E+09,8.999999E+09]];
    LOCAL CONST Robtarget Tr_meulage_motif_1_136 := [[20.52990625,142.768828125,26.117],[0.0569478960959874,-0.0562129652335629,0.700246962774789,-0.709402023393347],[0,0,0,0],[8.999999E+09,8.999999E+09,8.999999E+09,8.999999E+09,8.999999E+09,8.999999E+09]];
    LOCAL CONST Robtarget Tr_meulage_motif_1_137 := [[19.533810546875,142.68053125,26.116810546875],[0.0569478960959874,-0.0562129652335629,0.700246962774789,-0.709402023393347],[0,0,0,0],[8.999999E+09,8.999999E+09,8.999999E+09,8.999999E+09,8.999999E+09,8.999999E+09]];
    LOCAL CONST Robtarget Tr_meulage_motif_1_138 := [[18.545837890625,142.585078125,26.00630859375],[0.0569478960959874,-0.0562129652335629,0.700246962774789,-0.709402023393347],[0,0,0,0],[8.999999E+09,8.999999E+09,8.999999E+09,8.999999E+09,8.999999E+09,8.999999E+09]];
    LOCAL CONST Robtarget Tr_meulage_motif_1_139 := [[17.604396484375,142.486609375,25.79547265625],[0.0569478960959874,-0.0562129652335629,0.700246962774789,-0.709402023393347],[0,0,0,0],[8.999999E+09,8.999999E+09,8.999999E+09,8.999999E+09,8.999999E+09,8.999999E+09]];
    LOCAL CONST Robtarget Tr_meulage_motif_1_140 := [[16.756759765625,142.392125,25.52415234375],[0.0569478960959874,-0.0562129652335629,0.700246962774789,-0.709402023393347],[0,0,0,0],[8.999999E+09,8.999999E+09,8.999999E+09,8.999999E+09,8.999999E+09,8.999999E+09]];
    LOCAL CONST Robtarget Tr_meulage_motif_1_141 := [[16.01153125,142.3064375,25.248767578125],[0.0569478960959874,-0.0562129652335629,0.700246962774789,-0.709402023393347],[0,0,0,0],[8.999999E+09,8.999999E+09,8.999999E+09,8.999999E+09,8.999999E+09,8.999999E+09]];
    LOCAL CONST Robtarget Tr_meulage_motif_1_142 := [[14.9187412109375,142.16571875,24.633984375],[0.0569478960959874,-0.0562129652335629,0.700246962774789,-0.709402023393347],[0,0,0,0],[8.999999E+09,8.999999E+09,8.999999E+09,8.999999E+09,8.999999E+09,8.999999E+09]];
    LOCAL CONST Robtarget Tr_meulage_motif_1_143 := [[13.9043291015625,142.015484375,23.788265625],[0.0569478960959874,-0.0562129652335629,0.700246962774789,-0.709402023393347],[0,0,0,0],[8.999999E+09,8.999999E+09,8.999999E+09,8.999999E+09,8.999999E+09,8.999999E+09]];
    LOCAL CONST Robtarget Tr_meulage_motif_1_144 := [[13.066583984375,141.868359375,22.766806640625],[0.0569478960959874,-0.0562129652335629,0.700246962774789,-0.709402023393347],[0,0,0,0],[8.999999E+09,8.999999E+09,8.999999E+09,8.999999E+09,8.999999E+09,8.999999E+09]];
    LOCAL CONST Robtarget Tr_meulage_motif_1_145 := [[12.5875302734375,141.746453125,21.653333984375],[0.0569478960959874,-0.0562129652335629,0.700246962774789,-0.709402023393347],[0,0,0,0],[8.999999E+09,8.999999E+09,8.999999E+09,8.999999E+09,8.999999E+09,8.999999E+09]];
    LOCAL CONST Robtarget Tr_meulage_motif_1_146 := [[12.565060546875,141.6949375,20.959111328125],[0.0569478960959874,-0.0562129652335629,0.700246962774789,-0.709402023393347],[0,0,0,0],[8.999999E+09,8.999999E+09,8.999999E+09,8.999999E+09,8.999999E+09,8.999999E+09]];
    LOCAL CONST Robtarget Tr_meulage_motif_1_147 := [[12.5693232421875,141.64825,20.299525390625],[0.0569478960959874,-0.0562129652335629,0.700246962774789,-0.709402023393347],[0,0,0,0],[8.999999E+09,8.999999E+09,8.999999E+09,8.999999E+09,8.999999E+09,8.999999E+09]];
    LOCAL CONST Robtarget Tr_meulage_motif_1_148 := [[12.62824609375,141.6064375,19.64010546875],[0.0569478960959874,-0.0562129652335629,0.700246962774789,-0.709402023393347],[0,0,0,0],[8.999999E+09,8.999999E+09,8.999999E+09,8.999999E+09,8.999999E+09,8.999999E+09]];
    LOCAL CONST Robtarget Tr_meulage_motif_1_149 := [[13.1316220703125,141.572640625,18.541220703125],[0.0569478960959874,-0.0562129652335629,0.700246962774789,-0.709402023393347],[0,0,0,0],[8.999999E+09,8.999999E+09,8.999999E+09,8.999999E+09,8.999999E+09,8.999999E+09]];
    LOCAL CONST Robtarget Tr_meulage_motif_1_150 := [[13.991390625,141.57721875,17.537291015625],[0.0569478960959874,-0.0562129652335629,0.700246962774789,-0.709402023393347],[0,0,0,0],[8.999999E+09,8.999999E+09,8.999999E+09,8.999999E+09,8.999999E+09,8.999999E+09]];
    LOCAL CONST Robtarget Tr_meulage_motif_1_151 := [[15.0161435546875,141.6090625,16.710693359375],[0.0569478960959874,-0.0562129652335629,0.700246962774789,-0.709402023393347],[0,0,0,0],[8.999999E+09,8.999999E+09,8.999999E+09,8.999999E+09,8.999999E+09,8.999999E+09]];
    LOCAL CONST Robtarget Tr_meulage_motif_1_152 := [[15.7031044921875,141.641796875,16.3160693359375],[0.0569478960959874,-0.0562129652335629,0.700246962774789,-0.709402023393347],[0,0,0,0],[8.999999E+09,8.999999E+09,8.999999E+09,8.999999E+09,8.999999E+09,8.999999E+09]];
    LOCAL CONST Robtarget Tr_meulage_motif_1_153 := [[16.859880859375,141.709640625,15.8299833984375],[0.0569478960959874,-0.0562129652335629,0.700246962774789,-0.709402023393347],[0,0,0,0],[8.999999E+09,8.999999E+09,8.999999E+09,8.999999E+09,8.999999E+09,8.999999E+09]];
    LOCAL CONST Robtarget Tr_meulage_motif_1_154 := [[17.703314453125,141.765609375,15.5667138671875],[0.0569478960959874,-0.0562129652335629,0.700246962774789,-0.709402023393347],[0,0,0,0],[8.999999E+09,8.999999E+09,8.999999E+09,8.999999E+09,8.999999E+09,8.999999E+09]];
    LOCAL CONST Robtarget Tr_meulage_motif_1_155 := [[18.6329921875,141.83346875,15.362935546875],[0.0569478960959874,-0.0562129652335629,0.700246962774789,-0.709402023393347],[0,0,0,0],[8.999999E+09,8.999999E+09,8.999999E+09,8.999999E+09,8.999999E+09,8.999999E+09]];
    LOCAL CONST Robtarget Tr_meulage_motif_1_156 := [[19.611421875,141.91246875,15.25480078125],[0.0569478960959874,-0.0562129652335629,0.700246962774789,-0.709402023393347],[0,0,0,0],[8.999999E+09,8.999999E+09,8.999999E+09,8.999999E+09,8.999999E+09,8.999999E+09]];
    LOCAL CONST Robtarget Tr_meulage_motif_1_157 := [[20.6008203125,141.992296875,15.1446728515625],[0.0569478960959874,-0.0562129652335629,0.700246962774789,-0.709402023393347],[0,0,0,0],[8.999999E+09,8.999999E+09,8.999999E+09,8.999999E+09,8.999999E+09,8.999999E+09]];
    LOCAL CONST Robtarget Tr_meulage_motif_1_158 := [[21.5969140625,142.080578125,15.1448623046875],[0.0569478960959874,-0.0562129652335629,0.700246962774789,-0.709402023393347],[0,0,0,0],[8.999999E+09,8.999999E+09,8.999999E+09,8.999999E+09,8.999999E+09,8.999999E+09]];
    LOCAL CONST Robtarget Tr_meulage_motif_1_159 := [[22.593009765625,142.168875,15.14505078125],[0.0569478960959874,-0.0562129652335629,0.700246962774789,-0.709402023393347],[0,0,0,0],[8.999999E+09,8.999999E+09,8.999999E+09,8.999999E+09,8.999999E+09,8.999999E+09]];
    LOCAL CONST Robtarget Tr_meulage_motif_1_160 := [[23.589103515625,142.257171875,15.145240234375],[0.0569478960959874,-0.0562129652335629,0.700246962774789,-0.709402023393347],[0,0,0,0],[8.999999E+09,8.999999E+09,8.999999E+09,8.999999E+09,8.999999E+09,8.999999E+09]];
    LOCAL CONST Robtarget Tr_meulage_motif_1_161 := [[24.585197265625,142.34546875,15.1454287109375],[0.0569478960959874,-0.0562129652335629,0.700246962774789,-0.709402023393347],[0,0,0,0],[8.999999E+09,8.999999E+09,8.999999E+09,8.999999E+09,8.999999E+09,8.999999E+09]];
    LOCAL CONST Robtarget Tr_meulage_motif_1_162 := [[25.58129296875,142.433765625,15.1456181640625],[0.0569478960959874,-0.0562129652335629,0.700246962774789,-0.709402023393347],[0,0,0,0],[8.999999E+09,8.999999E+09,8.999999E+09,8.999999E+09,8.999999E+09,8.999999E+09]];
    LOCAL CONST Robtarget Tr_meulage_motif_1_163 := [[26.57738671875,142.5220625,15.1458076171875],[0.0569478960959874,-0.0562129652335629,0.700246962774789,-0.709402023393347],[0,0,0,0],[8.999999E+09,8.999999E+09,8.999999E+09,8.999999E+09,8.999999E+09,8.999999E+09]];
    LOCAL CONST Robtarget Tr_meulage_motif_1_164 := [[27.57348046875,142.61034375,15.14599609375],[0.0569478960959874,-0.0562129652335629,0.700246962774789,-0.709402023393347],[0,0,0,0],[8.999999E+09,8.999999E+09,8.999999E+09,8.999999E+09,8.999999E+09,8.999999E+09]];
    LOCAL CONST Robtarget Tr_meulage_motif_1_165 := [[28.569576171875,142.698640625,15.146185546875],[0.0569478960959874,-0.0562129652335629,0.700246962774789,-0.709402023393347],[0,0,0,0],[8.999999E+09,8.999999E+09,8.999999E+09,8.999999E+09,8.999999E+09,8.999999E+09]];
    LOCAL CONST Robtarget Tr_meulage_motif_1_166 := [[29.565669921875,142.7869375,15.1463740234375],[0.0569478960959874,-0.0562129652335629,0.700246962774789,-0.709402023393347],[0,0,0,0],[8.999999E+09,8.999999E+09,8.999999E+09,8.999999E+09,8.999999E+09,8.999999E+09]];
    LOCAL CONST Robtarget Tr_meulage_motif_1_167 := [[30.561765625,142.875234375,15.1465634765625],[0.0569478960959874,-0.0562129652335629,0.700246962774789,-0.709402023393347],[0,0,0,0],[8.999999E+09,8.999999E+09,8.999999E+09,8.999999E+09,8.999999E+09,8.999999E+09]];
    LOCAL CONST Robtarget Tr_meulage_motif_1_168 := [[31.557859375,142.96353125,15.1467529296875],[0.0569478960959874,-0.0562129652335629,0.700246962774789,-0.709402023393347],[0,0,0,0],[8.999999E+09,8.999999E+09,8.999999E+09,8.999999E+09,8.999999E+09,8.999999E+09]];
    LOCAL CONST Robtarget Tr_meulage_motif_1_169 := [[32.553953125,143.051828125,15.14694140625],[0.0569478960959874,-0.0562129652335629,0.700246962774789,-0.709402023393347],[0,0,0,0],[8.999999E+09,8.999999E+09,8.999999E+09,8.999999E+09,8.999999E+09,8.999999E+09]];
    LOCAL CONST Robtarget Tr_meulage_motif_1_170 := [[33.550046875,143.140109375,15.147130859375],[0.0569478960959874,-0.0562129652335629,0.700246962774789,-0.709402023393347],[0,0,0,0],[8.999999E+09,8.999999E+09,8.999999E+09,8.999999E+09,8.999999E+09,8.999999E+09]];
    LOCAL CONST Robtarget Tr_meulage_motif_1_171 := [[34.546140625,143.22840625,15.1473193359375],[0.0569478960959874,-0.0562129652335629,0.700246962774789,-0.709402023393347],[0,0,0,0],[8.999999E+09,8.999999E+09,8.999999E+09,8.999999E+09,8.999999E+09,8.999999E+09]];
    LOCAL CONST Robtarget Tr_meulage_motif_1_172 := [[35.54223828125,143.316703125,15.1475087890625],[0.0569478960959874,-0.0562129652335629,0.700246962774789,-0.709402023393347],[0,0,0,0],[8.999999E+09,8.999999E+09,8.999999E+09,8.999999E+09,8.999999E+09,8.999999E+09]];
    LOCAL CONST Robtarget Tr_meulage_motif_1_173 := [[36.53833203125,143.405,15.1476982421875],[0.0569478960959874,-0.0562129652335629,0.700246962774789,-0.709402023393347],[0,0,0,0],[8.999999E+09,8.999999E+09,8.999999E+09,8.999999E+09,8.999999E+09,8.999999E+09]];
    LOCAL CONST Robtarget Tr_meulage_motif_1_174 := [[37.53442578125,143.493296875,15.14788671875],[0.0569478960959874,-0.0562129652335629,0.700246962774789,-0.709402023393347],[0,0,0,0],[8.999999E+09,8.999999E+09,8.999999E+09,8.999999E+09,8.999999E+09,8.999999E+09]];
    LOCAL CONST Robtarget Tr_meulage_motif_1_175 := [[38.53051953125,143.58159375,15.148076171875],[0.0569478960959874,-0.0562129652335629,0.700246962774789,-0.709402023393347],[0,0,0,0],[8.999999E+09,8.999999E+09,8.999999E+09,8.999999E+09,8.999999E+09,8.999999E+09]];
    LOCAL CONST Robtarget Tr_meulage_motif_1_176 := [[39.52661328125,143.669875,15.1482646484375],[0.0569478960959874,-0.0562129652335629,0.700246962774789,-0.709402023393347],[0,0,0,0],[8.999999E+09,8.999999E+09,8.999999E+09,8.999999E+09,8.999999E+09,8.999999E+09]];
    LOCAL CONST Robtarget Tr_meulage_motif_1_177 := [[40.52270703125,143.758171875,15.1484541015625],[0.0569478960959874,-0.0562129652335629,0.700246962774789,-0.709402023393347],[0,0,0,0],[8.999999E+09,8.999999E+09,8.999999E+09,8.999999E+09,8.999999E+09,8.999999E+09]];
    LOCAL CONST Robtarget Tr_meulage_motif_1_178 := [[41.5188046875,143.84646875,15.148642578125],[0.0569478960959874,-0.0562129652335629,0.700246962774789,-0.709402023393347],[0,0,0,0],[8.999999E+09,8.999999E+09,8.999999E+09,8.999999E+09,8.999999E+09,8.999999E+09]];
    LOCAL CONST Robtarget Tr_meulage_motif_1_179 := [[42.5148984375,143.934765625,15.14883203125],[0.0569478960959874,-0.0562129652335629,0.700246962774789,-0.709402023393347],[0,0,0,0],[8.999999E+09,8.999999E+09,8.999999E+09,8.999999E+09,8.999999E+09,8.999999E+09]];
    LOCAL CONST Robtarget Tr_meulage_motif_1_180 := [[43.5109921875,144.0230625,15.149021484375],[0.0569478960959874,-0.0562129652335629,0.700246962774789,-0.709402023393347],[0,0,0,0],[8.999999E+09,8.999999E+09,8.999999E+09,8.999999E+09,8.999999E+09,8.999999E+09]];
    LOCAL CONST Robtarget Tr_meulage_motif_1_181 := [[44.5070859375,144.111359375,15.1492099609375],[0.0569478960959874,-0.0562129652335629,0.700246962774789,-0.709402023393347],[0,0,0,0],[8.999999E+09,8.999999E+09,8.999999E+09,8.999999E+09,8.999999E+09,8.999999E+09]];
    LOCAL CONST Robtarget Tr_meulage_motif_1_182 := [[45.5031796875,144.199640625,15.1493994140625],[0.0569478960959874,-0.0562129652335629,0.700246962774789,-0.709402023393347],[0,0,0,0],[8.999999E+09,8.999999E+09,8.999999E+09,8.999999E+09,8.999999E+09,8.999999E+09]];
    LOCAL CONST Robtarget Tr_meulage_motif_1_183 := [[46.49927734375,144.2879375,15.149587890625],[0.0569478960959874,-0.0562129652335629,0.700246962774789,-0.709402023393347],[0,0,0,0],[8.999999E+09,8.999999E+09,8.999999E+09,8.999999E+09,8.999999E+09,8.999999E+09]];
    LOCAL CONST Robtarget Tr_meulage_motif_1_184 := [[47.49537109375,144.376234375,15.14977734375],[0.0569478960959874,-0.0562129652335629,0.700246962774789,-0.709402023393347],[0,0,0,0],[8.999999E+09,8.999999E+09,8.999999E+09,8.999999E+09,8.999999E+09,8.999999E+09]];
    LOCAL CONST Robtarget Tr_meulage_motif_1_185 := [[48.49146484375,144.46453125,15.149966796875],[0.0569478960959874,-0.0562129652335629,0.700246962774789,-0.709402023393347],[0,0,0,0],[8.999999E+09,8.999999E+09,8.999999E+09,8.999999E+09,8.999999E+09,8.999999E+09]];
    LOCAL CONST Robtarget Tr_meulage_motif_1_186 := [[49.48755859375,144.552828125,15.1501552734375],[0.0569478960959874,-0.0562129652335629,0.700246962774789,-0.709402023393347],[0,0,0,0],[8.999999E+09,8.999999E+09,8.999999E+09,8.999999E+09,8.999999E+09,8.999999E+09]];
    LOCAL CONST Robtarget Tr_meulage_motif_1_187 := [[50.48365234375,144.641125,15.1503447265625],[0.0569478960959874,-0.0562129652335629,0.700246962774789,-0.709402023393347],[0,0,0,0],[8.999999E+09,8.999999E+09,8.999999E+09,8.999999E+09,8.999999E+09,8.999999E+09]];
    LOCAL CONST Robtarget Tr_meulage_motif_1_188 := [[51.47305078125,144.720953125,15.040216796875],[0.0569478960959874,-0.0562129652335629,0.700246962774789,-0.709402023393347],[0,0,0,0],[8.999999E+09,8.999999E+09,8.999999E+09,8.999999E+09,8.999999E+09,8.999999E+09]];
    LOCAL CONST Robtarget Tr_meulage_motif_1_189 := [[52.41721875,144.789609375,14.8297392578125],[0.0569478960959874,-0.0562129652335629,0.700246962774789,-0.709402023393347],[0,0,0,0],[8.999999E+09,8.999999E+09,8.999999E+09,8.999999E+09,8.999999E+09,8.999999E+09]];
    LOCAL CONST Robtarget Tr_meulage_motif_1_190 := [[53.268359375,144.845703125,14.558740234375],[0.0569478960959874,-0.0562129652335629,0.700246962774789,-0.709402023393347],[0,0,0,0],[8.999999E+09,8.999999E+09,8.999999E+09,8.999999E+09,8.999999E+09,8.999999E+09]];
    LOCAL CONST Robtarget Tr_meulage_motif_1_191 := [[53.9790390625,144.8870625,14.2555],[0.0569478960959874,-0.0562129652335629,0.700246962774789,-0.709402023393347],[0,0,0,0],[8.999999E+09,8.999999E+09,8.999999E+09,8.999999E+09,8.999999E+09,8.999999E+09]];
    LOCAL CONST Robtarget Tr_meulage_motif_1_192 := [[55.01373828125,144.931625,13.5948310546875],[0.0569478960959874,-0.0562129652335629,0.700246962774789,-0.709402023393347],[0,0,0,0],[8.999999E+09,8.999999E+09,8.999999E+09,8.999999E+09,8.999999E+09,8.999999E+09]];
    LOCAL CONST Robtarget Tr_meulage_motif_1_193 := [[55.91796875,144.94759375,12.6953173828125],[0.0569478960959874,-0.0562129652335629,0.700246962774789,-0.709402023393347],[0,0,0,0],[8.999999E+09,8.999999E+09,8.999999E+09,8.999999E+09,8.999999E+09,8.999999E+09]];
    LOCAL CONST Robtarget Tr_meulage_motif_1_194 := [[56.45759375,144.920984375,11.6520341796875],[0.0569478960959874,-0.0562129652335629,0.700246962774789,-0.709402023393347],[0,0,0,0],[8.999999E+09,8.999999E+09,8.999999E+09,8.999999E+09,8.999999E+09,8.999999E+09]];
    LOCAL CONST Robtarget Tr_meulage_motif_1_195 := [[56.64612109375,144.888359375,10.9605791015625],[0.0569478960959874,-0.0562129652335629,0.700246962774789,-0.709402023393347],[0,0,0,0],[8.999999E+09,8.999999E+09,8.999999E+09,8.999999E+09,8.999999E+09,8.999999E+09]];
    LOCAL CONST Robtarget Tr_meulage_motif_1_196 := [[56.7146796875,144.839640625,10.19252734375],[0.0569478960959874,-0.0562129652335629,0.700246962774789,-0.709402023393347],[0,0,0,0],[8.999999E+09,8.999999E+09,8.999999E+09,8.999999E+09,8.999999E+09,8.999999E+09]];
    LOCAL CONST Robtarget Tr_meulage_motif_1_197 := [[56.65296484375,144.779375,9.4245927734375],[0.0569478960959874,-0.0562129652335629,0.700246962774789,-0.709402023393347],[0,0,0,0],[8.999999E+09,8.999999E+09,8.999999E+09,8.999999E+09,8.999999E+09,8.999999E+09]];
    LOCAL CONST Robtarget Tr_meulage_motif_1_198 := [[56.24215625,144.66409375,8.31905078125],[0.0569478960959874,-0.0562129652335629,0.700246962774789,-0.709402023393347],[0,0,0,0],[8.999999E+09,8.999999E+09,8.999999E+09,8.999999E+09,8.999999E+09,8.999999E+09]];
    LOCAL CONST Robtarget Tr_meulage_motif_1_199 := [[55.83323828125,144.586171875,7.7347587890625],[0.0569478960959874,-0.0562129652335629,0.700246962774789,-0.709402023393347],[0,0,0,0],[8.999999E+09,8.999999E+09,8.999999E+09,8.999999E+09,8.999999E+09,8.999999E+09]];
    LOCAL CONST Robtarget Tr_meulage_motif_1_200 := [[54.955296875,144.44521875,6.84966650390625],[0.0569478960959874,-0.0562129652335629,0.700246962774789,-0.709402023393347],[0,0,0,0],[8.999999E+09,8.999999E+09,8.999999E+09,8.999999E+09,8.999999E+09,8.999999E+09]];
    LOCAL CONST Robtarget Tr_meulage_motif_1_201 := [[54.37456640625,144.36425,6.43631689453125],[0.0569478960959874,-0.0562129652335629,0.700246962774789,-0.709402023393347],[0,0,0,0],[8.999999E+09,8.999999E+09,8.999999E+09,8.999999E+09,8.999999E+09,8.999999E+09]];
    LOCAL CONST Robtarget Tr_meulage_motif_1_202 := [[53.26453515625,144.227140625,5.89334912109375],[0.0569478960959874,-0.0562129652335629,0.700246962774789,-0.709402023393347],[0,0,0,0],[8.999999E+09,8.999999E+09,8.999999E+09,8.999999E+09,8.999999E+09,8.999999E+09]];
    LOCAL CONST Robtarget Tr_meulage_motif_1_203 := [[52.4440703125,144.133390625,5.5984365234375],[0.0569478960959874,-0.0562129652335629,0.700246962774789,-0.709402023393347],[0,0,0,0],[8.999999E+09,8.999999E+09,8.999999E+09,8.999999E+09,8.999999E+09,8.999999E+09]];
    LOCAL CONST Robtarget Tr_meulage_motif_1_204 := [[51.51702734375,144.03665625,5.39429052734375],[0.0569478960959874,-0.0562129652335629,0.700246962774789,-0.709402023393347],[0,0,0,0],[8.999999E+09,8.999999E+09,8.999999E+09,8.999999E+09,8.999999E+09,8.999999E+09]];
    LOCAL CONST Robtarget Tr_meulage_motif_1_205 := [[50.54,143.942328125,5.2858310546875],[0.0569478960959874,-0.0562129652335629,0.700246962774789,-0.709402023393347],[0,0,0,0],[8.999999E+09,8.999999E+09,8.999999E+09,8.999999E+09,8.999999E+09,8.999999E+09]];
    LOCAL CONST Robtarget Tr_meulage_motif_1_206 := [[49.55202734375,143.846890625,5.1753125],[0.0569478960959874,-0.0562129652335629,0.700246962774789,-0.709402023393347],[0,0,0,0],[8.999999E+09,8.999999E+09,8.999999E+09,8.999999E+09,8.999999E+09,8.999999E+09]];
    LOCAL CONST Robtarget Tr_meulage_motif_1_207 := [[48.55593359375,143.75859375,5.175123046875],[0.0569478960959874,-0.0562129652335629,0.700246962774789,-0.709402023393347],[0,0,0,0],[8.999999E+09,8.999999E+09,8.999999E+09,8.999999E+09,8.999999E+09,8.999999E+09]];
    LOCAL CONST Robtarget Tr_meulage_motif_1_208 := [[47.5598359375,143.670296875,5.17493408203125],[0.0569478960959874,-0.0562129652335629,0.700246962774789,-0.709402023393347],[0,0,0,0],[8.999999E+09,8.999999E+09,8.999999E+09,8.999999E+09,8.999999E+09,8.999999E+09]];
    LOCAL CONST Robtarget Tr_meulage_motif_1_209 := [[46.5637421875,143.582,5.1747451171875],[0.0569478960959874,-0.0562129652335629,0.700246962774789,-0.709402023393347],[0,0,0,0],[8.999999E+09,8.999999E+09,8.999999E+09,8.999999E+09,8.999999E+09,8.999999E+09]];
    LOCAL CONST Robtarget Tr_meulage_motif_1_210 := [[45.5676484375,143.493703125,5.17455615234375],[0.0569478960959874,-0.0562129652335629,0.700246962774789,-0.709402023393347],[0,0,0,0],[8.999999E+09,8.999999E+09,8.999999E+09,8.999999E+09,8.999999E+09,8.999999E+09]];
    LOCAL CONST Robtarget Tr_meulage_motif_1_211 := [[44.5715546875,143.405421875,5.1743671875],[0.0569478960959874,-0.0562129652335629,0.700246962774789,-0.709402023393347],[0,0,0,0],[8.999999E+09,8.999999E+09,8.999999E+09,8.999999E+09,8.999999E+09,8.999999E+09]];
    LOCAL CONST Robtarget Tr_meulage_motif_1_212 := [[43.5754609375,143.317125,5.17417822265625],[0.0569478960959874,-0.0562129652335629,0.700246962774789,-0.709402023393347],[0,0,0,0],[8.999999E+09,8.999999E+09,8.999999E+09,8.999999E+09,8.999999E+09,8.999999E+09]];
    LOCAL CONST Robtarget Tr_meulage_motif_1_213 := [[42.5793671875,143.228828125,5.17398876953125],[0.0569478960959874,-0.0562129652335629,0.700246962774789,-0.709402023393347],[0,0,0,0],[8.999999E+09,8.999999E+09,8.999999E+09,8.999999E+09,8.999999E+09,8.999999E+09]];
    LOCAL CONST Robtarget Tr_meulage_motif_1_214 := [[41.58326953125,143.14053125,5.1737998046875],[0.0569478960959874,-0.0562129652335629,0.700246962774789,-0.709402023393347],[0,0,0,0],[8.999999E+09,8.999999E+09,8.999999E+09,8.999999E+09,8.999999E+09,8.999999E+09]];
    LOCAL CONST Robtarget Tr_meulage_motif_1_215 := [[40.58717578125,143.052234375,5.17361083984375],[0.0569478960959874,-0.0562129652335629,0.700246962774789,-0.709402023393347],[0,0,0,0],[8.999999E+09,8.999999E+09,8.999999E+09,8.999999E+09,8.999999E+09,8.999999E+09]];
    LOCAL CONST Robtarget Tr_meulage_motif_1_216 := [[39.59108203125,142.9639375,5.173421875],[0.0569478960959874,-0.0562129652335629,0.700246962774789,-0.709402023393347],[0,0,0,0],[8.999999E+09,8.999999E+09,8.999999E+09,8.999999E+09,8.999999E+09,8.999999E+09]];
    LOCAL CONST Robtarget Tr_meulage_motif_1_217 := [[38.59498828125,142.87565625,5.17323291015625],[0.0569478960959874,-0.0562129652335629,0.700246962774789,-0.709402023393347],[0,0,0,0],[8.999999E+09,8.999999E+09,8.999999E+09,8.999999E+09,8.999999E+09,8.999999E+09]];
    LOCAL CONST Robtarget Tr_meulage_motif_1_218 := [[37.59889453125,142.787359375,5.17304345703125],[0.0569478960959874,-0.0562129652335629,0.700246962774789,-0.709402023393347],[0,0,0,0],[8.999999E+09,8.999999E+09,8.999999E+09,8.999999E+09,8.999999E+09,8.999999E+09]];
    LOCAL CONST Robtarget Tr_meulage_motif_1_219 := [[36.60280078125,142.6990625,5.1728544921875],[0.0569478960959874,-0.0562129652335629,0.700246962774789,-0.709402023393347],[0,0,0,0],[8.999999E+09,8.999999E+09,8.999999E+09,8.999999E+09,8.999999E+09,8.999999E+09]];
    LOCAL CONST Robtarget Tr_meulage_motif_1_220 := [[35.606703125,142.610765625,5.17266552734375],[0.0569478960959874,-0.0562129652335629,0.700246962774789,-0.709402023393347],[0,0,0,0],[8.999999E+09,8.999999E+09,8.999999E+09,8.999999E+09,8.999999E+09,8.999999E+09]];
    LOCAL CONST Robtarget Tr_meulage_motif_1_221 := [[34.610609375,142.52246875,5.1724765625],[0.0569478960959874,-0.0562129652335629,0.700246962774789,-0.709402023393347],[0,0,0,0],[8.999999E+09,8.999999E+09,8.999999E+09,8.999999E+09,8.999999E+09,8.999999E+09]];
    LOCAL CONST Robtarget Tr_meulage_motif_1_222 := [[33.614515625,142.434171875,5.17228759765625],[0.0569478960959874,-0.0562129652335629,0.700246962774789,-0.709402023393347],[0,0,0,0],[8.999999E+09,8.999999E+09,8.999999E+09,8.999999E+09,8.999999E+09,8.999999E+09]];
    LOCAL CONST Robtarget Tr_meulage_motif_1_223 := [[32.618421875,142.345890625,5.1720986328125],[0.0569478960959874,-0.0562129652335629,0.700246962774789,-0.709402023393347],[0,0,0,0],[8.999999E+09,8.999999E+09,8.999999E+09,8.999999E+09,8.999999E+09,8.999999E+09]];
    LOCAL CONST Robtarget Tr_meulage_motif_1_224 := [[31.622326171875,142.25759375,5.1719091796875],[0.0569478960959874,-0.0562129652335629,0.700246962774789,-0.709402023393347],[0,0,0,0],[8.999999E+09,8.999999E+09,8.999999E+09,8.999999E+09,8.999999E+09,8.999999E+09]];
    LOCAL CONST Robtarget Tr_meulage_motif_1_225 := [[30.626232421875,142.169296875,5.17172021484375],[0.0569478960959874,-0.0562129652335629,0.700246962774789,-0.709402023393347],[0,0,0,0],[8.999999E+09,8.999999E+09,8.999999E+09,8.999999E+09,8.999999E+09,8.999999E+09]];
    LOCAL CONST Robtarget Tr_meulage_motif_1_226 := [[29.630138671875,142.081,5.17153125],[0.0569478960959874,-0.0562129652335629,0.700246962774789,-0.709402023393347],[0,0,0,0],[8.999999E+09,8.999999E+09,8.999999E+09,8.999999E+09,8.999999E+09,8.999999E+09]];
    LOCAL CONST Robtarget Tr_meulage_motif_1_227 := [[28.63404296875,141.992703125,5.17134228515625],[0.0569478960959874,-0.0562129652335629,0.700246962774789,-0.709402023393347],[0,0,0,0],[8.999999E+09,8.999999E+09,8.999999E+09,8.999999E+09,8.999999E+09,8.999999E+09]];
    LOCAL CONST Robtarget Tr_meulage_motif_1_228 := [[27.63794921875,141.90440625,5.1711533203125],[0.0569478960959874,-0.0562129652335629,0.700246962774789,-0.709402023393347],[0,0,0,0],[8.999999E+09,8.999999E+09,8.999999E+09,8.999999E+09,8.999999E+09,8.999999E+09]];
    LOCAL CONST Robtarget Tr_meulage_motif_1_229 := [[26.64185546875,141.816125,5.1709638671875],[0.0569478960959874,-0.0562129652335629,0.700246962774789,-0.709402023393347],[0,0,0,0],[8.999999E+09,8.999999E+09,8.999999E+09,8.999999E+09,8.999999E+09,8.999999E+09]];
    LOCAL CONST Robtarget Tr_meulage_motif_1_230 := [[25.645759765625,141.727828125,5.17077490234375],[0.0569478960959874,-0.0562129652335629,0.700246962774789,-0.709402023393347],[0,0,0,0],[8.999999E+09,8.999999E+09,8.999999E+09,8.999999E+09,8.999999E+09,8.999999E+09]];
    LOCAL CONST Robtarget Tr_meulage_motif_1_231 := [[24.649666015625,141.63953125,5.1705859375],[0.0569478960959874,-0.0562129652335629,0.700246962774789,-0.709402023393347],[0,0,0,0],[8.999999E+09,8.999999E+09,8.999999E+09,8.999999E+09,8.999999E+09,8.999999E+09]];
    LOCAL CONST Robtarget Tr_meulage_motif_1_232 := [[23.653572265625,141.551234375,5.17039697265625],[0.0569478960959874,-0.0562129652335629,0.700246962774789,-0.709402023393347],[0,0,0,0],[8.999999E+09,8.999999E+09,8.999999E+09,8.999999E+09,8.999999E+09,8.999999E+09]];
    LOCAL CONST Robtarget Tr_meulage_motif_1_233 := [[22.6574765625,141.4629375,5.1702080078125],[0.0569478960959874,-0.0562129652335629,0.700246962774789,-0.709402023393347],[0,0,0,0],[8.999999E+09,8.999999E+09,8.999999E+09,8.999999E+09,8.999999E+09,8.999999E+09]];
    LOCAL CONST Robtarget Tr_meulage_motif_1_234 := [[21.6613828125,141.374640625,5.17001904296875],[0.0569478960959874,-0.0562129652335629,0.700246962774789,-0.709402023393347],[0,0,0,0],[8.999999E+09,8.999999E+09,8.999999E+09,8.999999E+09,8.999999E+09,8.999999E+09]];
    LOCAL CONST Robtarget Tr_meulage_motif_1_235 := [[20.6652890625,141.286359375,5.16982958984375],[0.0569478960959874,-0.0562129652335629,0.700246962774789,-0.709402023393347],[0,0,0,0],[8.999999E+09,8.999999E+09,8.999999E+09,8.999999E+09,8.999999E+09,8.999999E+09]];
    LOCAL CONST Robtarget Tr_meulage_motif_1_236 := [[19.669193359375,141.1980625,5.169640625],[0.0569478960959874,-0.0562129652335629,0.700246962774789,-0.709402023393347],[0,0,0,0],[8.999999E+09,8.999999E+09,8.999999E+09,8.999999E+09,8.999999E+09,8.999999E+09]];
    LOCAL CONST Robtarget Tr_meulage_motif_1_237 := [[18.681220703125,141.102609375,5.0591220703125],[0.0569478960959874,-0.0562129652335629,0.700246962774789,-0.709402023393347],[0,0,0,0],[8.999999E+09,8.999999E+09,8.999999E+09,8.999999E+09,8.999999E+09,8.999999E+09]];
    LOCAL CONST Robtarget Tr_meulage_motif_1_238 := [[17.739779296875,141.004140625,4.84828662109375],[0.0569478960959874,-0.0562129652335629,0.700246962774789,-0.709402023393347],[0,0,0,0],[8.999999E+09,8.999999E+09,8.999999E+09,8.999999E+09,8.999999E+09,8.999999E+09]];
    LOCAL CONST Robtarget Tr_meulage_motif_1_239 := [[16.892142578125,140.90965625,4.5769814453125],[0.0569478960959874,-0.0562129652335629,0.700246962774789,-0.709402023393347],[0,0,0,0],[8.999999E+09,8.999999E+09,8.999999E+09,8.999999E+09,8.999999E+09,8.999999E+09]];
    LOCAL CONST Robtarget Tr_meulage_motif_1_240 := [[16.1853828125,140.825359375,4.27347119140625],[0.0569478960959874,-0.0562129652335629,0.700246962774789,-0.709402023393347],[0,0,0,0],[8.999999E+09,8.999999E+09,8.999999E+09,8.999999E+09,8.999999E+09,8.999999E+09]];
    LOCAL CONST Robtarget Tr_meulage_motif_1_241 := [[15.1592255859375,140.68725,3.6124111328125],[0.0569478960959874,-0.0562129652335629,0.700246962774789,-0.709402023393347],[0,0,0,0],[8.999999E+09,8.999999E+09,8.999999E+09,8.999999E+09,8.999999E+09,8.999999E+09]];
    LOCAL CONST Robtarget Tr_meulage_motif_1_242 := [[14.355583984375,140.549140625,2.67484033203125],[0.0569478960959874,-0.0562129652335629,0.700246962774789,-0.709402023393347],[0,0,0,0],[8.999999E+09,8.999999E+09,8.999999E+09,8.999999E+09,8.999999E+09,8.999999E+09]];
    LOCAL CONST Robtarget Tr_meulage_motif_1_243 := [[14.0109462890625,140.4476875,1.68092102050781],[0.0569478960959874,-0.0562129652335629,0.700246962774789,-0.709402023393347],[0,0,0,0],[8.999999E+09,8.999999E+09,8.999999E+09,8.999999E+09,8.999999E+09,8.999999E+09]];
    LOCAL CONST Robtarget Tr_meulage_motif_1_244 := [[14.0440810546875,140.4109375,1.12478234863281],[0.0569478960959874,-0.0562129652335629,0.700246962774789,-0.709402023393347],[0,0,0,0],[8.999999E+09,8.999999E+09,8.999999E+09,8.999999E+09,8.999999E+09,8.999999E+09]];
    LOCAL CONST Robtarget Tr_meulage_motif_1_245 := [[14.0424794921875,140.3810625,0.707926574707031],[0.0569478960959874,-0.0562129652335629,0.700246962774789,-0.709402023393347],[0,0,0,0],[8.999999E+09,8.999999E+09,8.999999E+09,8.999999E+09,8.999999E+09,8.999999E+09]];
    LOCAL CONST Robtarget Tr_meulage_motif_1_246 := [[14.4094697265625,140.344609375,-0.258894561767578],[0.0569478960959874,-0.0562129652335629,0.700246962774789,-0.709402023393347],[0,0,0,0],[8.999999E+09,8.999999E+09,8.999999E+09,8.999999E+09,8.999999E+09,8.999999E+09]];
    LOCAL CONST Robtarget Tr_meulage_motif_1_247 := [[15.23411328125,140.35240625,-1.17411804199219],[0.0569478960959874,-0.0562129652335629,0.700246962774789,-0.709402023393347],[0,0,0,0],[8.999999E+09,8.999999E+09,8.999999E+09,8.999999E+09,8.999999E+09,8.999999E+09]];
    LOCAL CONST Robtarget Tr_meulage_motif_1_248 := [[15.84660546875,140.37659375,-1.5958291015625],[0.0569478960959874,-0.0562129652335629,0.700246962774789,-0.709402023393347],[0,0,0,0],[8.999999E+09,8.999999E+09,8.999999E+09,8.999999E+09,8.999999E+09,8.999999E+09]];
    LOCAL CONST Robtarget Tr_meulage_motif_1_249 := [[16.975923828125,140.438953125,-2.12473413085938],[0.0569478960959874,-0.0562129652335629,0.700246962774789,-0.709402023393347],[0,0,0,0],[8.999999E+09,8.999999E+09,8.999999E+09,8.999999E+09,8.999999E+09,8.999999E+09]];
    LOCAL CONST Robtarget Tr_meulage_motif_1_250 := [[17.81935546875,140.494921875,-2.38801928710937],[0.0569478960959874,-0.0562129652335629,0.700246962774789,-0.709402023393347],[0,0,0,0],[8.999999E+09,8.999999E+09,8.999999E+09,8.999999E+09,8.999999E+09,8.999999E+09]];
    LOCAL CONST Robtarget Tr_meulage_motif_1_251 := [[18.74903515625,140.562765625,-2.59181298828125],[0.0569478960959874,-0.0562129652335629,0.700246962774789,-0.709402023393347],[0,0,0,0],[8.999999E+09,8.999999E+09,8.999999E+09,8.999999E+09,8.999999E+09,8.999999E+09]];
    LOCAL CONST Robtarget Tr_meulage_motif_1_252 := [[19.727462890625,140.64178125,-2.6999013671875],[0.0569478960959874,-0.0562129652335629,0.700246962774789,-0.709402023393347],[0,0,0,0],[8.999999E+09,8.999999E+09,8.999999E+09,8.999999E+09,8.999999E+09,8.999999E+09]];
    LOCAL CONST Robtarget Tr_meulage_motif_1_253 := [[20.71686328125,140.721609375,-2.81004467773438],[0.0569478960959874,-0.0562129652335629,0.700246962774789,-0.709402023393347],[0,0,0,0],[8.999999E+09,8.999999E+09,8.999999E+09,8.999999E+09,8.999999E+09,8.999999E+09]];
    LOCAL CONST Robtarget Tr_meulage_motif_1_254 := [[21.71295703125,140.809890625,-2.80985571289062],[0.0569478960959874,-0.0562129652335629,0.700246962774789,-0.709402023393347],[0,0,0,0],[8.999999E+09,8.999999E+09,8.999999E+09,8.999999E+09,8.999999E+09,8.999999E+09]];
    LOCAL CONST Robtarget Tr_meulage_motif_1_255 := [[22.70905078125,140.8981875,-2.80966674804688],[0.0569478960959874,-0.0562129652335629,0.700246962774789,-0.709402023393347],[0,0,0,0],[8.999999E+09,8.999999E+09,8.999999E+09,8.999999E+09,8.999999E+09,8.999999E+09]];
    LOCAL CONST Robtarget Tr_meulage_motif_1_256 := [[23.705146484375,140.986484375,-2.8094775390625],[0.0569478960959874,-0.0562129652335629,0.700246962774789,-0.709402023393347],[0,0,0,0],[8.999999E+09,8.999999E+09,8.999999E+09,8.999999E+09,8.999999E+09,8.999999E+09]];
    LOCAL CONST Robtarget Tr_meulage_motif_1_257 := [[24.701240234375,141.07478125,-2.80928857421875],[0.0569478960959874,-0.0562129652335629,0.700246962774789,-0.709402023393347],[0,0,0,0],[8.999999E+09,8.999999E+09,8.999999E+09,8.999999E+09,8.999999E+09,8.999999E+09]];
    LOCAL CONST Robtarget Tr_meulage_motif_1_258 := [[25.697333984375,141.163078125,-2.80909936523437],[0.0569478960959874,-0.0562129652335629,0.700246962774789,-0.709402023393347],[0,0,0,0],[8.999999E+09,8.999999E+09,8.999999E+09,8.999999E+09,8.999999E+09,8.999999E+09]];
    LOCAL CONST Robtarget Tr_meulage_motif_1_259 := [[26.6934296875,141.251375,-2.80891040039063],[0.0569478960959874,-0.0562129652335629,0.700246962774789,-0.709402023393347],[0,0,0,0],[8.999999E+09,8.999999E+09,8.999999E+09,8.999999E+09,8.999999E+09,8.999999E+09]];
    LOCAL CONST Robtarget Tr_meulage_motif_1_260 := [[27.6895234375,141.33965625,-2.80872143554688],[0.0569478960959874,-0.0562129652335629,0.700246962774789,-0.709402023393347],[0,0,0,0],[8.999999E+09,8.999999E+09,8.999999E+09,8.999999E+09,8.999999E+09,8.999999E+09]];
    LOCAL CONST Robtarget Tr_meulage_motif_1_261 := [[28.6856171875,141.427953125,-2.8085322265625],[0.0569478960959874,-0.0562129652335629,0.700246962774789,-0.709402023393347],[0,0,0,0],[8.999999E+09,8.999999E+09,8.999999E+09,8.999999E+09,8.999999E+09,8.999999E+09]];
    LOCAL CONST Robtarget Tr_meulage_motif_1_262 := [[29.681712890625,141.51625,-2.80834326171875],[0.0569478960959874,-0.0562129652335629,0.700246962774789,-0.709402023393347],[0,0,0,0],[8.999999E+09,8.999999E+09,8.999999E+09,8.999999E+09,8.999999E+09,8.999999E+09]];
    LOCAL CONST Robtarget Tr_meulage_motif_1_263 := [[30.677806640625,141.604546875,-2.808154296875],[0.0569478960959874,-0.0562129652335629,0.700246962774789,-0.709402023393347],[0,0,0,0],[8.999999E+09,8.999999E+09,8.999999E+09,8.999999E+09,8.999999E+09,8.999999E+09]];
    LOCAL CONST Robtarget Tr_meulage_motif_1_264 := [[31.673900390625,141.69284375,-2.80796508789063],[0.0569478960959874,-0.0562129652335629,0.700246962774789,-0.709402023393347],[0,0,0,0],[8.999999E+09,8.999999E+09,8.999999E+09,8.999999E+09,8.999999E+09,8.999999E+09]];
    LOCAL CONST Robtarget Tr_meulage_motif_1_265 := [[32.66999609375,141.781140625,-2.80777612304687],[0.0569478960959874,-0.0562129652335629,0.700246962774789,-0.709402023393347],[0,0,0,0],[8.999999E+09,8.999999E+09,8.999999E+09,8.999999E+09,8.999999E+09,8.999999E+09]];
    LOCAL CONST Robtarget Tr_meulage_motif_1_266 := [[33.66608984375,141.869421875,-2.80758715820313],[0.0569478960959874,-0.0562129652335629,0.700246962774789,-0.709402023393347],[0,0,0,0],[8.999999E+09,8.999999E+09,8.999999E+09,8.999999E+09,8.999999E+09,8.999999E+09]];
    LOCAL CONST Robtarget Tr_meulage_motif_1_267 := [[34.66218359375,141.95771875,-2.80739794921875],[0.0569478960959874,-0.0562129652335629,0.700246962774789,-0.709402023393347],[0,0,0,0],[8.999999E+09,8.999999E+09,8.999999E+09,8.999999E+09,8.999999E+09,8.999999E+09]];
    LOCAL CONST Robtarget Tr_meulage_motif_1_268 := [[35.65827734375,142.046015625,-2.807208984375],[0.0569478960959874,-0.0562129652335629,0.700246962774789,-0.709402023393347],[0,0,0,0],[8.999999E+09,8.999999E+09,8.999999E+09,8.999999E+09,8.999999E+09,8.999999E+09]];
    LOCAL CONST Robtarget Tr_meulage_motif_1_269 := [[36.654375,142.1343125,-2.80701977539062],[0.0569478960959874,-0.0562129652335629,0.700246962774789,-0.709402023393347],[0,0,0,0],[8.999999E+09,8.999999E+09,8.999999E+09,8.999999E+09,8.999999E+09,8.999999E+09]];
    LOCAL CONST Robtarget Tr_meulage_motif_1_270 := [[37.65046875,142.222609375,-2.80683081054688],[0.0569478960959874,-0.0562129652335629,0.700246962774789,-0.709402023393347],[0,0,0,0],[8.999999E+09,8.999999E+09,8.999999E+09,8.999999E+09,8.999999E+09,8.999999E+09]];
    LOCAL CONST Robtarget Tr_meulage_motif_1_271 := [[38.6465625,142.31090625,-2.80664184570313],[0.0569478960959874,-0.0562129652335629,0.700246962774789,-0.709402023393347],[0,0,0,0],[8.999999E+09,8.999999E+09,8.999999E+09,8.999999E+09,8.999999E+09,8.999999E+09]];
    LOCAL CONST Robtarget Tr_meulage_motif_1_272 := [[39.64265625,142.3991875,-2.80645263671875],[0.0569478960959874,-0.0562129652335629,0.700246962774789,-0.709402023393347],[0,0,0,0],[8.999999E+09,8.999999E+09,8.999999E+09,8.999999E+09,8.999999E+09,8.999999E+09]];
    LOCAL CONST Robtarget Tr_meulage_motif_1_273 := [[40.63875,142.487484375,-2.806263671875],[0.0569478960959874,-0.0562129652335629,0.700246962774789,-0.709402023393347],[0,0,0,0],[8.999999E+09,8.999999E+09,8.999999E+09,8.999999E+09,8.999999E+09,8.999999E+09]];
    LOCAL CONST Robtarget Tr_meulage_motif_1_274 := [[41.63484375,142.57578125,-2.80607470703125],[0.0569478960959874,-0.0562129652335629,0.700246962774789,-0.709402023393347],[0,0,0,0],[8.999999E+09,8.999999E+09,8.999999E+09,8.999999E+09,8.999999E+09,8.999999E+09]];
    LOCAL CONST Robtarget Tr_meulage_motif_1_275 := [[42.63094140625,142.664078125,-2.80588549804688],[0.0569478960959874,-0.0562129652335629,0.700246962774789,-0.709402023393347],[0,0,0,0],[8.999999E+09,8.999999E+09,8.999999E+09,8.999999E+09,8.999999E+09,8.999999E+09]];
    LOCAL CONST Robtarget Tr_meulage_motif_1_276 := [[43.62703515625,142.752375,-2.80569653320312],[0.0569478960959874,-0.0562129652335629,0.700246962774789,-0.709402023393347],[0,0,0,0],[8.999999E+09,8.999999E+09,8.999999E+09,8.999999E+09,8.999999E+09,8.999999E+09]];
    LOCAL CONST Robtarget Tr_meulage_motif_1_277 := [[44.62312890625,142.84065625,-2.80550756835938],[0.0569478960959874,-0.0562129652335629,0.700246962774789,-0.709402023393347],[0,0,0,0],[8.999999E+09,8.999999E+09,8.999999E+09,8.999999E+09,8.999999E+09,8.999999E+09]];
    LOCAL CONST Robtarget Tr_meulage_motif_1_278 := [[45.61922265625,142.928953125,-2.805318359375],[0.0569478960959874,-0.0562129652335629,0.700246962774789,-0.709402023393347],[0,0,0,0],[8.999999E+09,8.999999E+09,8.999999E+09,8.999999E+09,8.999999E+09,8.999999E+09]];
    LOCAL CONST Robtarget Tr_meulage_motif_1_279 := [[46.61531640625,143.01725,-2.80512939453125],[0.0569478960959874,-0.0562129652335629,0.700246962774789,-0.709402023393347],[0,0,0,0],[8.999999E+09,8.999999E+09,8.999999E+09,8.999999E+09,8.999999E+09,8.999999E+09]];
    LOCAL CONST Robtarget Tr_meulage_motif_1_280 := [[47.61141015625,143.105546875,-2.80494018554687],[0.0569478960959874,-0.0562129652335629,0.700246962774789,-0.709402023393347],[0,0,0,0],[8.999999E+09,8.999999E+09,8.999999E+09,8.999999E+09,8.999999E+09,8.999999E+09]];
    LOCAL CONST Robtarget Tr_meulage_motif_1_281 := [[48.6075078125,143.19384375,-2.80475122070313],[0.0569478960959874,-0.0562129652335629,0.700246962774789,-0.709402023393347],[0,0,0,0],[8.999999E+09,8.999999E+09,8.999999E+09,8.999999E+09,8.999999E+09,8.999999E+09]];
    LOCAL CONST Robtarget Tr_meulage_motif_1_282 := [[49.6036015625,143.282140625,-2.80456225585938],[0.0569478960959874,-0.0562129652335629,0.700246962774789,-0.709402023393347],[0,0,0,0],[8.999999E+09,8.999999E+09,8.999999E+09,8.999999E+09,8.999999E+09,8.999999E+09]];
    LOCAL CONST Robtarget Tr_meulage_motif_1_283 := [[50.5996953125,143.370421875,-2.804373046875],[0.0569478960959874,-0.0562129652335629,0.700246962774789,-0.709402023393347],[0,0,0,0],[8.999999E+09,8.999999E+09,8.999999E+09,8.999999E+09,8.999999E+09,8.999999E+09]];
    LOCAL CONST Robtarget Tr_meulage_motif_1_284 := [[51.5957890625,143.45871875,-2.80418408203125],[0.0569478960959874,-0.0562129652335629,0.700246962774789,-0.709402023393347],[0,0,0,0],[8.999999E+09,8.999999E+09,8.999999E+09,8.999999E+09,8.999999E+09,8.999999E+09]];
    LOCAL CONST Robtarget Tr_meulage_motif_1_285 := [[52.5918828125,143.547015625,-2.8039951171875],[0.0569478960959874,-0.0562129652335629,0.700246962774789,-0.709402023393347],[0,0,0,0],[8.999999E+09,8.999999E+09,8.999999E+09,8.999999E+09,8.999999E+09,8.999999E+09]];
    LOCAL CONST Robtarget Tr_meulage_motif_1_286 := [[53.5879765625,143.6353125,-2.80380590820313],[0.0569478960959874,-0.0562129652335629,0.700246962774789,-0.709402023393347],[0,0,0,0],[8.999999E+09,8.999999E+09,8.999999E+09,8.999999E+09,8.999999E+09,8.999999E+09]];
    LOCAL CONST Robtarget Tr_meulage_motif_1_287 := [[54.58407421875,143.723609375,-2.80361694335937],[0.0569478960959874,-0.0562129652335629,0.700246962774789,-0.709402023393347],[0,0,0,0],[8.999999E+09,8.999999E+09,8.999999E+09,8.999999E+09,8.999999E+09,8.999999E+09]];
    LOCAL CONST Robtarget Tr_meulage_motif_1_288 := [[55.58016796875,143.81190625,-2.80342797851563],[0.0569478960959874,-0.0562129652335629,0.700246962774789,-0.709402023393347],[0,0,0,0],[8.999999E+09,8.999999E+09,8.999999E+09,8.999999E+09,8.999999E+09,8.999999E+09]];
    LOCAL CONST Robtarget Tr_meulage_motif_1_289 := [[56.57626171875,143.9001875,-2.80323876953125],[0.0569478960959874,-0.0562129652335629,0.700246962774789,-0.709402023393347],[0,0,0,0],[8.999999E+09,8.999999E+09,8.999999E+09,8.999999E+09,8.999999E+09,8.999999E+09]];
    LOCAL CONST Robtarget Tr_meulage_motif_1_290 := [[57.57235546875,143.988484375,-2.8030498046875],[0.0569478960959874,-0.0562129652335629,0.700246962774789,-0.709402023393347],[0,0,0,0],[8.999999E+09,8.999999E+09,8.999999E+09,8.999999E+09,8.999999E+09,8.999999E+09]];
    LOCAL CONST Robtarget Tr_meulage_motif_1_291 := [[58.56844921875,144.07678125,-2.80286059570312],[0.0569478960959874,-0.0562129652335629,0.700246962774789,-0.709402023393347],[0,0,0,0],[8.999999E+09,8.999999E+09,8.999999E+09,8.999999E+09,8.999999E+09,8.999999E+09]];
    LOCAL CONST Robtarget Tr_meulage_motif_1_292 := [[59.564546875,144.165078125,-2.80267163085938],[0.0569478960959874,-0.0562129652335629,0.700246962774789,-0.709402023393347],[0,0,0,0],[8.999999E+09,8.999999E+09,8.999999E+09,8.999999E+09,8.999999E+09,8.999999E+09]];
    LOCAL CONST Robtarget Tr_meulage_motif_1_293 := [[60.560640625,144.253375,-2.80248266601563],[0.0569478960959874,-0.0562129652335629,0.700246962774789,-0.709402023393347],[0,0,0,0],[8.999999E+09,8.999999E+09,8.999999E+09,8.999999E+09,8.999999E+09,8.999999E+09]];
    LOCAL CONST Robtarget Tr_meulage_motif_1_294 := [[61.556734375,144.341671875,-2.80229345703125],[0.0569478960959874,-0.0562129652335629,0.700246962774789,-0.709402023393347],[0,0,0,0],[8.999999E+09,8.999999E+09,8.999999E+09,8.999999E+09,8.999999E+09,8.999999E+09]];

